C07313=1137.764,345.073,-80.303,-176.559,9.353,148.899
C07314=1137.768,344.825,-80.268,-176.562,9.349,148.898
C07315=1137.772,344.578,-80.235,-176.564,9.345,148.898
C07316=1137.777,344.331,-80.200,-176.567,9.341,148.898
C07317=1137.780,344.083,-80.166,-176.569,9.337,148.897
C07318=1137.784,343.836,-80.131,-176.572,9.333,148.897
C07319=1137.788,343.588,-80.097,-176.574,9.329,148.897
C07320=1137.792,343.340,-80.063,-176.577,9.325,148.896
C07321=1137.796,343.092,-80.029,-176.579,9.321,148.896
C07322=1137.800,342.844,-79.995,-176.582,9.318,148.896
C07323=1137.805,342.597,-79.960,-176.584,9.313,148.895
C07324=1137.808,342.349,-79.926,-176.587,9.309,148.895
C07325=1137.813,342.102,-79.891,-176.590,9.305,148.895
C07326=1137.816,341.854,-79.857,-176.592,9.301,148.894
C07327=1137.820,341.607,-79.823,-176.595,9.297,148.894
C07328=1137.825,341.359,-79.790,-176.597,9.293,148.894
C07329=1137.828,341.111,-79.755,-176.600,9.290,148.893
C07330=1137.832,340.864,-79.721,-176.602,9.285,148.893
C07331=1137.836,340.617,-79.687,-176.605,9.281,148.893
C07332=1137.840,340.368,-79.652,-176.607,9.278,148.892
C07333=1137.844,340.121,-79.619,-176.610,9.274,148.892
C07334=1137.849,339.873,-79.585,-176.613,9.270,148.892
C07335=1137.852,339.625,-79.550,-176.615,9.266,148.891
C07336=1137.857,339.345,-79.512,-176.618,9.261,148.891
C07337=1137.862,339.064,-79.473,-176.621,9.257,148.891
C07338=1137.866,338.783,-79.435,-176.624,9.253,148.891
C07339=1137.870,338.502,-79.396,-176.626,9.248,148.890
C07340=1137.875,338.255,-79.363,-176.629,9.244,148.890
C07341=1137.878,338.007,-79.329,-176.632,9.240,148.890
C07342=1137.882,337.759,-79.294,-176.634,9.237,148.889
C07343=1137.887,337.512,-79.261,-176.637,9.233,148.889
C07344=1137.890,337.265,-79.227,-176.640,9.228,148.889
C07345=1137.894,337.016,-79.194,-176.642,9.225,148.888
C07346=1137.899,336.769,-79.159,-176.645,9.221,148.888
C07347=1137.903,336.521,-79.126,-176.648,9.217,148.888
C07348=1137.906,336.274,-79.092,-176.650,9.213,148.887
C07349=1137.910,336.025,-79.059,-176.653,9.209,148.887
C07350=1137.915,335.778,-79.024,-176.655,9.206,148.887
C07351=1137.919,335.530,-78.991,-176.658,9.201,148.887
C07352=1137.923,335.283,-78.957,-176.660,9.197,148.886
C07353=1137.926,335.035,-78.924,-176.663,9.194,148.886
C07354=1137.930,334.788,-78.890,-176.665,9.190,148.886
C07355=1137.935,334.540,-78.856,-176.668,9.186,148.885
C07356=1137.939,334.292,-78.822,-176.671,9.182,148.885
C07357=1137.942,334.044,-78.789,-176.673,9.178,148.885
C07358=1137.946,333.796,-78.755,-176.676,9.174,148.885
C07359=1137.950,333.549,-78.722,-176.678,9.171,148.884
C07360=1137.954,333.301,-78.688,-176.681,9.166,148.884
C07361=1137.959,333.053,-78.655,-176.683,9.163,148.884
C07362=1137.962,332.806,-78.620,-176.686,9.159,148.884
C07363=1137.967,332.558,-78.587,-176.689,9.155,148.883
C07364=1137.971,332.310,-78.554,-176.691,9.151,148.883
C07365=1137.975,332.062,-78.521,-176.694,9.147,148.883
C07366=1137.979,331.815,-78.487,-176.696,9.144,148.882
C07367=1137.982,331.567,-78.454,-176.699,9.140,148.882
C07368=1137.986,331.319,-78.420,-176.702,9.136,148.882
C07369=1137.990,331.071,-78.387,-176.704,9.132,148.882
C07370=1137.994,330.824,-78.353,-176.707,9.128,148.881
C07371=1137.998,330.577,-78.320,-176.709,9.125,148.881
C07372=1138.003,330.329,-78.287,-176.712,9.121,148.881
C07373=1138.007,330.081,-78.254,-176.715,9.117,148.880
C07374=1138.011,329.832,-78.220,-176.717,9.113,148.880
C07375=1138.015,329.585,-78.187,-176.720,9.109,148.880
C07376=1138.019,329.337,-78.153,-176.722,9.106,148.880
C07377=1138.023,329.089,-78.120,-176.725,9.102,148.879
C07378=1138.027,328.842,-78.088,-176.728,9.098,148.879
C07379=1138.031,328.595,-78.054,-176.730,9.094,148.879
C07380=1138.035,328.347,-78.021,-176.733,9.090,148.879
C07381=1138.039,328.099,-77.988,-176.735,9.087,148.878
C07382=1138.043,327.851,-77.954,-176.738,9.083,148.878
C07383=1138.047,327.604,-77.921,-176.740,9.079,148.878
C07384=1138.051,327.356,-77.888,-176.743,9.075,148.878
C07385=1138.055,327.108,-77.855,-176.746,9.071,148.877
C07386=1138.059,326.859,-77.822,-176.749,9.068,148.877
C07387=1138.063,326.612,-77.789,-176.751,9.063,148.877
C07388=1138.068,326.364,-77.756,-176.753,9.060,148.877
C07389=1138.072,326.116,-77.723,-176.756,9.056,148.876
C07390=1138.076,325.868,-77.690,-176.759,9.053,148.876
C07391=1138.079,325.621,-77.657,-176.762,9.049,148.876
C07392=1138.083,325.373,-77.624,-176.765,9.045,148.876
C07393=1138.088,325.125,-77.591,-176.767,9.042,148.876
C07394=1138.092,324.878,-77.557,-176.769,9.037,148.875
C07395=1138.096,324.629,-77.525,-176.772,9.034,148.875
C07396=1138.100,324.382,-77.492,-176.775,9.030,148.875
C07397=1138.104,324.134,-77.459,-176.777,9.027,148.875
C07398=1138.108,323.886,-77.426,-176.780,9.022,148.874
C07399=1138.112,323.638,-77.394,-176.782,9.019,148.874
C07400=1138.116,323.390,-77.361,-176.785,9.015,148.874
C07401=1138.120,323.143,-77.328,-176.788,9.011,148.874
C07402=1138.124,322.895,-77.295,-176.790,9.008,148.873
C07403=1138.128,322.647,-77.262,-176.793,9.003,148.873
C07404=1138.132,322.399,-77.229,-176.795,9.000,148.873
C07405=1138.136,322.152,-77.197,-176.798,8.996,148.873
C07406=1138.140,321.903,-77.164,-176.801,8.993,148.872
C07407=1138.144,321.656,-77.131,-176.804,8.989,148.872
C07408=1138.148,321.408,-77.099,-176.806,8.986,148.872
C07409=1138.153,321.161,-77.066,-176.809,8.981,148.872
C07410=1138.157,320.913,-77.033,-176.811,8.978,148.872
C07411=1138.161,320.665,-77.001,-176.814,8.974,148.871
C07412=1138.165,320.417,-76.968,-176.816,8.971,148.871
C07413=1138.169,320.169,-76.935,-176.819,8.967,148.871
C07414=1138.173,319.921,-76.903,-176.822,8.964,148.871
C07415=1138.177,319.674,-76.870,-176.825,8.959,148.871
C07416=1138.181,319.425,-76.838,-176.827,8.956,148.870
C07417=1138.185,319.178,-76.805,-176.830,8.952,148.870
C07418=1138.189,318.929,-76.773,-176.832,8.949,148.870
C07419=1138.193,318.682,-76.740,-176.835,8.945,148.870
C07420=1138.198,318.434,-76.708,-176.838,8.940,148.869
C07421=1138.201,318.186,-76.676,-176.840,8.937,148.869
C07422=1138.205,317.939,-76.643,-176.843,8.933,148.869
C07423=1138.210,317.690,-76.611,-176.845,8.930,148.869
C07424=1138.213,317.443,-76.578,-176.848,8.926,148.869
C07425=1138.218,317.195,-76.546,-176.851,8.923,148.868
C07426=1138.221,316.947,-76.514,-176.854,8.918,148.868
C07427=1138.226,316.699,-76.481,-176.856,8.915,148.868
C07428=1138.230,316.451,-76.449,-176.859,8.911,148.868
C07429=1138.234,316.203,-76.417,-176.862,8.908,148.868
C07430=1138.238,315.956,-76.384,-176.864,8.904,148.867
C07431=1138.242,315.707,-76.352,-176.867,8.901,148.867
C07432=1138.246,315.460,-76.320,-176.869,8.898,148.867
C07433=1138.251,315.212,-76.287,-176.872,8.894,148.867
C07434=1138.254,314.964,-76.255,-176.874,8.890,148.867
C07435=1138.259,314.716,-76.223,-176.877,8.886,148.867
C07436=1138.262,314.468,-76.191,-176.880,8.883,148.866
C07437=1138.267,314.220,-76.159,-176.883,8.879,148.866
C07438=1138.271,313.973,-76.126,-176.885,8.876,148.866
C07439=1138.275,313.725,-76.094,-176.888,8.872,148.866
C07440=1138.280,313.447,-76.058,-176.891,8.867,148.865
C07441=1138.284,313.169,-76.023,-176.894,8.863,148.865
C07442=1138.289,312.890,-75.987,-176.897,8.859,148.865
C07443=1138.294,312.612,-75.951,-176.900,8.855,148.865
C07444=1138.298,312.364,-75.919,-176.902,8.852,148.865
C07445=1138.302,312.117,-75.887,-176.905,8.848,148.864
C07446=1138.306,311.869,-75.854,-176.908,8.845,148.864
C07447=1138.310,311.621,-75.822,-176.911,8.841,148.864
C07448=1138.313,311.373,-75.790,-176.913,8.838,148.864
C07449=1138.318,311.126,-75.758,-176.916,8.834,148.864
C07450=1138.322,310.877,-75.727,-176.918,8.830,148.864
C07451=1138.326,310.629,-75.695,-176.921,8.826,148.863
C07452=1138.331,310.382,-75.663,-176.924,8.823,148.863
C07453=1138.335,310.134,-75.631,-176.926,8.819,148.863
C07454=1138.339,309.885,-75.600,-176.929,8.816,148.863
C07455=1138.343,309.638,-75.568,-176.932,8.813,148.863
C07456=1138.347,309.389,-75.536,-176.935,8.809,148.863
C07457=1138.351,309.141,-75.504,-176.937,8.805,148.862
C07458=1138.355,308.894,-75.472,-176.940,8.801,148.862
C07459=1138.359,308.646,-75.441,-176.942,8.798,148.862
C07460=1138.364,308.398,-75.408,-176.945,8.794,148.862
C07461=1138.368,308.150,-75.377,-176.947,8.791,148.862
C07462=1138.372,307.902,-75.345,-176.950,8.788,148.862
C07463=1138.376,307.654,-75.314,-176.953,8.784,148.861
C07464=1138.380,307.406,-75.282,-176.955,8.781,148.861
C07465=1138.384,307.158,-75.250,-176.958,8.776,148.861
C07466=1138.389,306.911,-75.218,-176.961,8.773,148.861
C07467=1138.393,306.662,-75.187,-176.964,8.769,148.861
C07468=1138.397,306.415,-75.156,-176.966,8.766,148.861
C07469=1138.401,306.167,-75.124,-176.969,8.763,148.861
C07470=1138.405,305.918,-75.093,-176.972,8.759,148.860
C07471=1138.409,305.671,-75.061,-176.974,8.756,148.860
C07472=1138.413,305.422,-75.029,-176.977,8.752,148.860
C07473=1138.418,305.175,-74.997,-176.980,8.749,148.860
C07474=1138.422,304.926,-74.966,-176.983,8.745,148.860
C07475=1138.426,304.679,-74.935,-176.985,8.741,148.860
C07476=1138.430,304.430,-74.904,-176.987,8.738,148.859
C07477=1138.434,304.183,-74.872,-176.990,8.734,148.859
C07478=1138.438,303.935,-74.840,-176.993,8.731,148.859
C07479=1138.443,303.687,-74.809,-176.996,8.727,148.859
C07480=1138.446,303.439,-74.778,-176.998,8.724,148.859
C07481=1138.451,303.191,-74.747,-177.001,8.720,148.859
C07482=1138.455,302.943,-74.715,-177.004,8.717,148.859
C07483=1138.459,302.695,-74.684,-177.006,8.713,148.858
C07484=1138.463,302.447,-74.652,-177.009,8.709,148.858
C07485=1138.468,302.199,-74.622,-177.012,8.706,148.858
C07486=1138.471,301.951,-74.590,-177.014,8.703,148.858
C07487=1138.476,301.703,-74.559,-177.017,8.699,148.858
C07488=1138.480,301.455,-74.527,-177.020,8.696,148.858
C07489=1138.484,301.207,-74.496,-177.023,8.692,148.858
C07490=1138.488,300.958,-74.465,-177.025,8.689,148.858
C07491=1138.493,300.711,-74.434,-177.028,8.686,148.857
C07492=1138.497,300.462,-74.403,-177.031,8.682,148.857
C07493=1138.501,300.215,-74.371,-177.033,8.678,148.857
C07494=1138.505,299.966,-74.340,-177.036,8.675,148.857
C07495=1138.510,299.718,-74.309,-177.039,8.671,148.857
C07496=1138.513,299.470,-74.277,-177.041,8.668,148.857
C07497=1138.518,299.222,-74.247,-177.045,8.664,148.857
C07498=1138.522,298.975,-74.216,-177.047,8.661,148.856
C07499=1138.525,298.727,-74.185,-177.049,8.658,148.856
C07500=1138.530,298.479,-74.154,-177.053,8.654,148.856
C07501=1138.534,298.230,-74.123,-177.055,8.651,148.856
C07502=1138.539,297.982,-74.092,-177.057,8.648,148.856
C07503=1138.543,297.735,-74.061,-177.060,8.643,148.856
C07504=1138.546,297.486,-74.030,-177.063,8.641,148.856
C07505=1138.551,297.238,-73.999,-177.066,8.636,148.856
C07506=1138.555,296.990,-73.968,-177.068,8.633,148.855
C07507=1138.559,296.742,-73.937,-177.071,8.630,148.855
C07508=1138.564,296.494,-73.907,-177.074,8.626,148.855
C07509=1138.567,296.246,-73.875,-177.076,8.623,148.855
C07510=1138.572,295.998,-73.845,-177.079,8.620,148.855
C07511=1138.576,295.750,-73.814,-177.082,8.616,148.855
C07512=1138.580,295.501,-73.783,-177.085,8.613,148.855
C07513=1138.584,295.254,-73.752,-177.087,8.610,148.855
C07514=1138.589,295.006,-73.722,-177.090,8.606,148.855
C07515=1138.593,294.757,-73.691,-177.093,8.603,148.855
C07516=1138.597,294.510,-73.660,-177.095,8.600,148.854
C07517=1138.601,294.262,-73.630,-177.098,8.595,148.854
C07518=1138.605,294.013,-73.599,-177.101,8.593,148.854
C07519=1138.610,293.765,-73.568,-177.103,8.589,148.854
C07520=1138.614,293.517,-73.538,-177.106,8.585,148.854
C07521=1138.618,293.269,-73.506,-177.109,8.582,148.854
C07522=1138.622,293.021,-73.476,-177.111,8.579,148.854
C07523=1138.626,292.773,-73.446,-177.115,8.575,148.854
C07524=1138.630,292.524,-73.414,-177.117,8.572,148.854
C07525=1138.634,292.277,-73.384,-177.119,8.569,148.853
C07526=1138.639,292.029,-73.353,-177.123,8.565,148.853
C07527=1138.643,291.781,-73.323,-177.125,8.562,148.853
C07528=1138.647,291.533,-73.292,-177.128,8.559,148.853
C07529=1138.652,291.284,-73.262,-177.131,8.555,148.853
C07530=1138.655,291.036,-73.232,-177.134,8.552,148.853
C07531=1138.660,290.788,-73.201,-177.136,8.549,148.853
C07532=1138.663,290.540,-73.171,-177.139,8.545,148.853
C07533=1138.668,290.292,-73.140,-177.142,8.542,148.853
C07534=1138.673,290.044,-73.109,-177.144,8.538,148.853
C07535=1138.677,289.796,-73.080,-177.147,8.535,148.853
C07536=1138.681,289.547,-73.049,-177.150,8.531,148.852
C07537=1138.685,289.299,-73.018,-177.152,8.528,148.853
C07538=1138.689,289.052,-72.988,-177.155,8.525,148.852
C07539=1138.693,288.803,-72.958,-177.158,8.521,148.852
C07540=1138.698,288.555,-72.927,-177.161,8.518,148.852
C07541=1138.701,288.307,-72.897,-177.163,8.515,148.852
C07542=1138.706,288.058,-72.867,-177.166,8.511,148.852
C07543=1138.710,287.811,-72.837,-177.169,8.508,148.852
C07544=1138.714,287.535,-72.803,-177.172,8.504,148.852
C07545=1138.720,287.260,-72.770,-177.174,8.501,148.852
C07546=1138.724,286.984,-72.736,-177.178,8.497,148.852
C07547=1138.729,286.709,-72.702,-177.181,8.493,148.852
C07548=1138.733,286.460,-72.672,-177.183,8.490,148.852
C07549=1138.737,286.212,-72.642,-177.186,8.486,148.851
C07550=1138.742,285.964,-72.612,-177.189,8.483,148.851
C07551=1138.746,285.716,-72.582,-177.191,8.480,148.851
C07552=1138.750,285.468,-72.552,-177.194,8.477,148.851
C07553=1138.754,285.220,-72.522,-177.197,8.473,148.851
C07554=1138.759,284.972,-72.492,-177.200,8.470,148.851
C07555=1138.763,284.724,-72.462,-177.202,8.467,148.851
C07556=1138.767,284.475,-72.432,-177.205,8.464,148.851
C07557=1138.771,284.227,-72.402,-177.208,8.460,148.851
C07558=1138.775,283.979,-72.371,-177.211,8.457,148.851
C07559=1138.780,283.730,-72.342,-177.213,8.454,148.851
C07560=1138.784,283.483,-72.312,-177.217,8.450,148.851
C07561=1138.788,283.234,-72.282,-177.219,8.447,148.851
C07562=1138.792,282.986,-72.252,-177.222,8.444,148.851
C07563=1138.797,282.738,-72.222,-177.224,8.440,148.850
C07564=1138.801,282.490,-72.192,-177.227,8.437,148.850
C07565=1138.805,282.242,-72.162,-177.230,8.434,148.850
C07566=1138.810,281.994,-72.133,-177.233,8.430,148.850
C07567=1138.814,281.745,-72.103,-177.235,8.428,148.850
C07568=1138.818,281.497,-72.072,-177.238,8.423,148.850
C07569=1138.822,281.249,-72.043,-177.241,8.421,148.850
C07570=1138.827,281.001,-72.013,-177.243,8.417,148.850
C07571=1138.831,280.753,-71.984,-177.246,8.414,148.850
C07572=1138.835,280.505,-71.954,-177.249,8.410,148.850
C07573=1138.840,280.256,-71.924,-177.252,8.407,148.850
C07574=1138.844,280.008,-71.894,-177.255,8.404,148.850
C07575=1138.848,279.760,-71.865,-177.257,8.401,148.850
C07576=1138.852,279.512,-71.835,-177.260,8.397,148.850
C07577=1138.856,279.264,-71.805,-177.263,8.394,148.850
C07578=1138.860,279.016,-71.776,-177.265,8.391,148.850
C07579=1138.864,278.767,-71.746,-177.268,8.388,148.850
C07580=1138.869,278.519,-71.716,-177.271,8.384,148.850
C07581=1138.874,278.271,-71.687,-177.274,8.381,148.850
C07582=1138.878,278.022,-71.657,-177.276,8.378,148.850
C07583=1138.882,277.774,-71.628,-177.279,8.375,148.850
C07584=1138.886,277.526,-71.598,-177.281,8.372,148.849
C07585=1138.890,277.277,-71.569,-177.285,8.368,148.849
C07586=1138.894,277.029,-71.540,-177.288,8.365,148.849
C07587=1138.899,276.781,-71.510,-177.290,8.362,148.849
C07588=1138.903,276.533,-71.481,-177.293,8.359,148.849
C07589=1138.907,276.284,-71.451,-177.296,8.355,148.849
C07590=1138.911,276.036,-71.422,-177.298,8.352,148.849
C07591=1138.915,275.788,-71.392,-177.301,8.349,148.849
C07592=1138.920,275.540,-71.363,-177.304,8.346,148.849
C07593=1138.924,275.292,-71.334,-177.306,8.343,148.849
C07594=1138.928,275.044,-71.304,-177.310,8.339,148.849
C07595=1138.933,274.795,-71.275,-177.312,8.336,148.849
C07596=1138.937,274.547,-71.245,-177.315,8.333,148.849
C07597=1138.941,274.299,-71.216,-177.318,8.330,148.849
C07598=1138.945,274.051,-71.186,-177.320,8.327,148.849
C07599=1138.949,273.802,-71.157,-177.323,8.323,148.849
C07600=1138.954,273.554,-71.129,-177.326,8.320,148.849
C07601=1138.959,273.306,-71.099,-177.329,8.317,148.849
C07602=1138.963,273.058,-71.070,-177.331,8.314,148.849
C07603=1138.967,272.809,-71.040,-177.334,8.311,148.849
C07604=1138.971,272.561,-71.011,-177.337,8.307,148.849
C07605=1138.976,272.312,-70.982,-177.340,8.304,148.849
C07606=1138.979,272.064,-70.953,-177.342,8.301,148.849
C07607=1138.984,271.817,-70.924,-177.345,8.298,148.849
C07608=1138.988,271.568,-70.895,-177.348,8.295,148.849
C07609=1138.993,271.320,-70.866,-177.351,8.291,148.849
C07610=1138.997,271.071,-70.836,-177.354,8.288,148.849
C07611=1139.001,270.823,-70.807,-177.356,8.285,148.849
C07612=1139.006,270.575,-70.779,-177.359,8.282,148.849
C07613=1139.009,270.327,-70.750,-177.361,8.279,148.849
C07614=1139.014,270.079,-70.720,-177.364,8.276,148.849
C07615=1139.018,269.830,-70.692,-177.368,8.272,148.849
C07616=1139.023,269.582,-70.663,-177.370,8.269,148.849
C07617=1139.027,269.333,-70.634,-177.373,8.266,148.849
C07618=1139.031,269.085,-70.605,-177.376,8.263,148.849
C07619=1139.035,268.837,-70.575,-177.378,8.260,148.849
C07620=1139.040,268.589,-70.547,-177.381,8.257,148.849
C07621=1139.044,268.341,-70.518,-177.384,8.253,148.849
C07622=1139.048,268.092,-70.489,-177.386,8.250,148.848
C07623=1139.052,267.844,-70.460,-177.389,8.247,148.849
C07624=1139.057,267.596,-70.432,-177.392,8.244,148.849
C07625=1139.062,267.347,-70.402,-177.395,8.241,148.849
C07626=1139.065,267.099,-70.374,-177.397,8.238,148.849
C07627=1139.070,266.851,-70.345,-177.400,8.234,148.849
C07628=1139.075,266.602,-70.316,-177.403,8.231,148.849
C07629=1139.078,266.354,-70.287,-177.406,8.228,148.849
C07630=1139.082,266.105,-70.259,-177.408,8.225,148.849
C07631=1139.088,265.857,-70.230,-177.411,8.222,148.849
C07632=1139.091,265.609,-70.201,-177.414,8.219,148.849
C07633=1139.095,265.360,-70.173,-177.417,8.216,148.849
C07634=1139.101,265.112,-70.144,-177.420,8.212,148.848
C07635=1139.104,264.864,-70.115,-177.422,8.209,148.849
C07636=1139.109,264.615,-70.087,-177.425,8.206,148.849
C07637=1139.113,264.368,-70.059,-177.428,8.204,148.849
C07638=1139.117,264.119,-70.029,-177.430,8.200,148.849
C07639=1139.122,263.871,-70.001,-177.433,8.197,148.849
C07640=1139.126,263.622,-69.973,-177.436,8.194,148.849
C07641=1139.130,263.374,-69.944,-177.439,8.191,148.849
C07642=1139.134,263.126,-69.916,-177.442,8.187,148.849
C07643=1139.139,262.877,-69.887,-177.445,8.185,148.849
C07644=1139.143,262.629,-69.858,-177.447,8.182,148.849
C07645=1139.147,262.381,-69.830,-177.450,8.179,148.849
C07646=1139.152,262.132,-69.801,-177.452,8.175,148.849
C07647=1139.156,261.885,-69.773,-177.455,8.173,148.849
C07648=1139.161,261.610,-69.742,-177.459,8.169,148.849
C07649=1139.166,261.337,-69.711,-177.461,8.166,148.849
C07650=1139.171,261.064,-69.679,-177.465,8.162,148.849
C07651=1139.175,260.790,-69.648,-177.468,8.159,148.849
C07652=1139.180,260.542,-69.620,-177.471,8.155,148.849
C07653=1139.184,260.293,-69.591,-177.473,8.152,148.849
C07654=1139.188,260.045,-69.564,-177.476,8.149,148.849
C07655=1139.193,259.796,-69.535,-177.479,8.146,148.849
C07656=1139.197,259.548,-69.507,-177.482,8.143,148.849
C07657=1139.201,259.300,-69.478,-177.484,8.141,148.849
C07658=1139.206,259.052,-69.451,-177.487,8.137,148.849
C07659=1139.210,258.803,-69.422,-177.490,8.134,148.849
C07660=1139.214,258.554,-69.394,-177.492,8.131,148.849
C07661=1139.218,258.306,-69.366,-177.496,8.128,148.849
C07662=1139.223,258.057,-69.337,-177.499,8.125,148.849
C07663=1139.227,257.810,-69.309,-177.501,8.122,148.849
C07664=1139.231,257.561,-69.281,-177.504,8.119,148.849
C07665=1139.236,257.313,-69.253,-177.507,8.116,148.849
C07666=1139.240,257.064,-69.225,-177.509,8.113,148.849
C07667=1139.244,256.816,-69.197,-177.512,8.110,148.849
C07668=1139.249,256.568,-69.169,-177.515,8.107,148.849
C07669=1139.253,256.320,-69.140,-177.517,8.104,148.849
C07670=1139.258,256.071,-69.113,-177.520,8.101,148.849
C07671=1139.262,255.822,-69.085,-177.523,8.098,148.849
C07672=1139.266,255.574,-69.057,-177.526,8.095,148.849
C07673=1139.270,255.326,-69.029,-177.529,8.091,148.849
C07674=1139.275,255.078,-69.000,-177.532,8.088,148.849
C07675=1139.279,254.829,-68.972,-177.535,8.085,148.849
C07676=1139.284,254.580,-68.945,-177.537,8.082,148.849
C07677=1139.288,254.333,-68.917,-177.540,8.079,148.849
C07678=1139.293,254.084,-68.889,-177.543,8.076,148.849
C07679=1139.297,253.836,-68.861,-177.545,8.073,148.850
C07680=1139.301,253.587,-68.833,-177.548,8.070,148.850
C07681=1139.305,253.339,-68.806,-177.551,8.068,148.850
C07682=1139.309,253.090,-68.778,-177.554,8.065,148.850
C07683=1139.314,252.841,-68.750,-177.557,8.062,148.850
C07684=1139.319,252.594,-68.722,-177.559,8.058,148.850
C07685=1139.323,252.345,-68.694,-177.562,8.056,148.850
C07686=1139.327,252.096,-68.667,-177.564,8.053,148.850
C07687=1139.332,251.849,-68.639,-177.567,8.050,148.850
C07688=1139.336,251.599,-68.612,-177.571,8.046,148.850
C07689=1139.341,251.351,-68.583,-177.573,8.043,148.850
C07690=1139.344,251.103,-68.555,-177.576,8.040,148.850
C07691=1139.349,250.854,-68.528,-177.579,8.037,148.850
C07692=1139.353,250.606,-68.500,-177.582,8.034,148.850
C07693=1139.358,250.357,-68.473,-177.584,8.031,148.850
C07694=1139.362,250.109,-68.445,-177.587,8.028,148.850
C07695=1139.367,249.861,-68.418,-177.590,8.025,148.850
C07696=1139.370,249.612,-68.390,-177.593,8.022,148.850
C07697=1139.375,249.364,-68.363,-177.595,8.019,148.850
C07698=1139.379,249.116,-68.335,-177.598,8.016,148.850
C07699=1139.383,248.867,-68.308,-177.601,8.014,148.851
C07700=1139.388,248.619,-68.280,-177.604,8.011,148.851
C07701=1139.392,248.370,-68.253,-177.607,8.008,148.851
C07702=1139.397,248.122,-68.224,-177.609,8.005,148.851
C07703=1139.401,247.873,-68.197,-177.612,8.002,148.851
C07704=1139.406,247.624,-68.170,-177.615,7.999,148.851
C07705=1139.410,247.376,-68.142,-177.617,7.996,148.851
C07706=1139.415,247.128,-68.115,-177.620,7.993,148.851
C07707=1139.419,246.879,-68.088,-177.623,7.990,148.851
C07708=1139.423,246.631,-68.061,-177.626,7.987,148.851
C07709=1139.427,246.383,-68.033,-177.628,7.984,148.851
C07710=1139.432,246.133,-68.006,-177.631,7.981,148.851
C07711=1139.436,245.886,-67.978,-177.634,7.978,148.851
C07712=1139.441,245.637,-67.951,-177.637,7.975,148.851
C07713=1139.445,245.389,-67.924,-177.640,7.972,148.851
C07714=1139.450,245.140,-67.897,-177.642,7.969,148.851
C07715=1139.454,244.891,-67.869,-177.645,7.967,148.851
C07716=1139.458,244.643,-67.842,-177.648,7.964,148.852
C07717=1139.463,244.395,-67.815,-177.651,7.961,148.852
C07718=1139.468,244.146,-67.788,-177.654,7.958,148.852
C07719=1139.472,243.898,-67.761,-177.656,7.955,148.852
C07720=1139.475,243.649,-67.733,-177.659,7.952,148.852
C07721=1139.480,243.401,-67.706,-177.662,7.949,148.852
C07722=1139.485,243.152,-67.679,-177.665,7.946,148.852
C07723=1139.489,242.904,-67.652,-177.668,7.943,148.852
C07724=1139.494,242.655,-67.625,-177.670,7.940,148.852
C07725=1139.498,242.406,-67.597,-177.673,7.937,148.852
C07726=1139.502,242.158,-67.571,-177.676,7.934,148.852
C07727=1139.506,241.909,-67.544,-177.679,7.932,148.852
C07728=1139.511,241.662,-67.516,-177.682,7.929,148.853
C07729=1139.516,241.413,-67.489,-177.684,7.926,148.853
C07730=1139.520,241.165,-67.462,-177.687,7.923,148.853
C07731=1139.524,240.916,-67.436,-177.690,7.920,148.853
C07732=1139.528,240.667,-67.408,-177.693,7.917,148.853
C07733=1139.533,240.419,-67.381,-177.696,7.914,148.853
C07734=1139.537,240.170,-67.354,-177.698,7.911,148.853
C07735=1139.541,239.922,-67.328,-177.701,7.908,148.853
C07736=1139.546,239.673,-67.301,-177.704,7.905,148.853
C07737=1139.551,239.424,-67.274,-177.707,7.902,148.853
C07738=1139.555,239.176,-67.248,-177.710,7.900,148.853
C07739=1139.560,238.928,-67.221,-177.712,7.897,148.853
C07740=1139.564,238.679,-67.194,-177.715,7.894,148.853
C07741=1139.568,238.431,-67.167,-177.718,7.891,148.854
C07742=1139.573,238.183,-67.140,-177.721,7.888,148.854
C07743=1139.577,237.933,-67.113,-177.724,7.885,148.854
C07744=1139.581,237.685,-67.086,-177.726,7.882,148.854
C07745=1139.586,237.436,-67.060,-177.729,7.879,148.854
C07746=1139.590,237.187,-67.033,-177.732,7.876,148.854
C07747=1139.594,236.939,-67.006,-177.735,7.873,148.854
C07748=1139.599,236.691,-66.979,-177.738,7.870,148.854
C07749=1139.604,236.442,-66.952,-177.740,7.867,148.854
C07750=1139.608,236.194,-66.926,-177.743,7.865,148.854
C07751=1139.613,235.945,-66.899,-177.746,7.862,148.854
C07752=1139.618,235.673,-66.870,-177.749,7.859,148.854
C07753=1139.622,235.402,-66.841,-177.752,7.856,148.855
C07754=1139.627,235.129,-66.812,-177.754,7.853,148.855
C07755=1139.632,234.858,-66.783,-177.758,7.850,148.855
C07756=1139.636,234.609,-66.756,-177.761,7.847,148.855
C07757=1139.641,234.360,-66.730,-177.764,7.844,148.855
C07758=1139.645,234.112,-66.704,-177.767,7.841,148.855
C07759=1139.649,233.864,-66.677,-177.769,7.838,148.855
C07760=1139.654,233.615,-66.651,-177.772,7.836,148.855
C07761=1139.658,233.366,-66.624,-177.774,7.833,148.855
C07762=1139.663,233.118,-66.598,-177.777,7.830,148.856
C07763=1139.667,232.869,-66.571,-177.780,7.827,148.856
C07764=1139.671,232.621,-66.544,-177.783,7.824,148.856
C07765=1139.676,232.372,-66.518,-177.786,7.821,148.856
C07766=1139.680,232.124,-66.492,-177.788,7.818,148.856
C07767=1139.685,231.874,-66.465,-177.791,7.815,148.856
C07768=1139.689,231.626,-66.439,-177.794,7.812,148.856
C07769=1139.694,231.378,-66.413,-177.797,7.810,148.856
C07770=1139.698,231.130,-66.386,-177.800,7.807,148.856
C07771=1139.703,230.881,-66.361,-177.803,7.804,148.856
C07772=1139.707,230.632,-66.334,-177.805,7.802,148.857
C07773=1139.711,230.384,-66.308,-177.808,7.799,148.857
C07774=1139.716,230.135,-66.282,-177.811,7.796,148.857
C07775=1139.720,229.886,-66.255,-177.814,7.793,148.857
C07776=1139.725,229.637,-66.229,-177.816,7.790,148.857
C07777=1139.729,229.389,-66.202,-177.819,7.787,148.857
C07778=1139.734,229.141,-66.177,-177.822,7.785,148.857
C07779=1139.738,228.892,-66.151,-177.825,7.782,148.857
C07780=1139.743,228.644,-66.124,-177.828,7.779,148.858
C07781=1139.747,228.395,-66.098,-177.831,7.776,148.858
C07782=1139.751,228.146,-66.072,-177.833,7.774,148.858
C07783=1139.756,227.897,-66.045,-177.836,7.771,148.858
C07784=1139.760,227.649,-66.020,-177.839,7.768,148.858
C07785=1139.765,227.401,-65.994,-177.841,7.765,148.858
C07786=1139.769,227.152,-65.968,-177.844,7.762,148.858
C07787=1139.774,226.903,-65.941,-177.847,7.760,148.858
C07788=1139.778,226.654,-65.916,-177.850,7.757,148.858
C07789=1139.782,226.406,-65.890,-177.853,7.754,148.859
C07790=1139.786,226.157,-65.863,-177.856,7.751,148.859
C07791=1139.792,225.909,-65.838,-177.858,7.749,148.859
C07792=1139.796,225.660,-65.812,-177.861,7.746,148.859
C07793=1139.800,225.411,-65.786,-177.864,7.743,148.859
C07794=1139.805,225.163,-65.760,-177.867,7.740,148.859
C07795=1139.810,224.915,-65.734,-177.870,7.738,148.859
C07796=1139.814,224.666,-65.708,-177.873,7.735,148.859
C07797=1139.818,224.417,-65.682,-177.875,7.732,148.860
C07798=1139.823,224.168,-65.656,-177.878,7.729,148.860
C07799=1139.827,223.920,-65.631,-177.880,7.727,148.860
C07800=1139.832,223.671,-65.605,-177.883,7.724,148.860
C07801=1139.837,223.422,-65.579,-177.887,7.721,148.860
C07802=1139.841,223.174,-65.553,-177.889,7.719,148.860
C07803=1139.845,222.925,-65.527,-177.892,7.716,148.860
C07804=1139.850,222.677,-65.502,-177.895,7.713,148.860
C07805=1139.854,222.428,-65.476,-177.898,7.710,148.861
C07806=1139.858,222.179,-65.450,-177.900,7.708,148.861
C07807=1139.863,221.931,-65.425,-177.903,7.705,148.861
C07808=1139.867,221.682,-65.399,-177.906,7.702,148.861
C07809=1139.872,221.433,-65.374,-177.909,7.699,148.861
C07810=1139.876,221.185,-65.348,-177.912,7.696,148.861
C07811=1139.881,220.936,-65.322,-177.914,7.694,148.861
C07812=1139.886,220.687,-65.296,-177.917,7.692,148.862
C07813=1139.890,220.439,-65.270,-177.920,7.689,148.862
C07814=1139.895,220.190,-65.245,-177.923,7.686,148.862
C07815=1139.899,219.942,-65.219,-177.926,7.683,148.862
C07816=1139.903,219.693,-65.193,-177.928,7.680,148.862
C07817=1139.908,219.445,-65.168,-177.932,7.678,148.862
C07818=1139.912,219.195,-65.143,-177.934,7.675,148.862
C07819=1139.917,218.946,-65.117,-177.937,7.673,148.863
C07820=1139.921,218.698,-65.092,-177.939,7.670,148.863
C07821=1139.926,218.450,-65.066,-177.942,7.667,148.863
C07822=1139.930,218.201,-65.041,-177.945,7.664,148.863
C07823=1139.935,217.952,-65.016,-177.948,7.662,148.863
C07824=1139.939,217.704,-64.991,-177.951,7.659,148.863
C07825=1139.943,217.455,-64.965,-177.953,7.656,148.863
C07826=1139.948,217.207,-64.939,-177.956,7.653,148.864
C07827=1139.952,216.957,-64.914,-177.959,7.651,148.864
C07828=1139.957,216.709,-64.889,-177.962,7.648,148.864
C07829=1139.961,216.460,-64.863,-177.964,7.646,148.864
C07830=1139.966,216.212,-64.838,-177.967,7.643,148.864
C07831=1139.970,215.963,-64.813,-177.970,7.640,148.864
C07832=1139.975,215.714,-64.787,-177.973,7.637,148.865
C07833=1139.980,215.466,-64.762,-177.976,7.635,148.865
C07834=1139.983,215.217,-64.737,-177.978,7.632,148.865
C07835=1139.988,214.969,-64.712,-177.982,7.630,148.865
C07836=1139.993,214.719,-64.687,-177.984,7.627,148.865
C07837=1139.998,214.471,-64.661,-177.987,7.624,148.865
C07838=1140.002,214.222,-64.636,-177.989,7.622,148.865
C07839=1140.007,213.974,-64.611,-177.993,7.619,148.866
C07840=1140.010,213.725,-64.586,-177.996,7.617,148.866
C07841=1140.015,213.476,-64.561,-177.998,7.614,148.866
C07842=1140.020,213.228,-64.535,-178.001,7.611,148.866
C07843=1140.024,212.978,-64.510,-178.004,7.609,148.866
C07844=1140.029,212.730,-64.485,-178.007,7.606,148.866
C07845=1140.033,212.481,-64.461,-178.009,7.603,148.867
C07846=1140.038,212.233,-64.435,-178.013,7.601,148.867
C07847=1140.042,211.983,-64.410,-178.015,7.599,148.867
C07848=1140.047,211.735,-64.385,-178.018,7.596,148.867
C07849=1140.051,211.486,-64.360,-178.021,7.593,148.867
C07850=1140.056,211.238,-64.335,-178.024,7.590,148.868
C07851=1140.060,210.989,-64.310,-178.027,7.587,148.868
C07852=1140.065,210.740,-64.286,-178.029,7.585,148.868
C07853=1140.069,210.492,-64.260,-178.032,7.583,148.868
C07854=1140.074,210.243,-64.235,-178.035,7.580,148.868
C07855=1140.079,209.995,-64.210,-178.038,7.577,148.868
C07856=1140.083,209.724,-64.183,-178.041,7.574,148.869
C07857=1140.088,209.453,-64.156,-178.044,7.571,148.869
C07858=1140.093,209.183,-64.129,-178.047,7.568,148.869
C07859=1140.098,208.912,-64.102,-178.050,7.566,148.869
C07860=1140.103,208.663,-64.077,-178.053,7.563,148.869
C07861=1140.107,208.414,-64.053,-178.055,7.561,148.869
C07862=1140.111,208.166,-64.028,-178.058,7.558,148.870
C07863=1140.116,207.917,-64.003,-178.061,7.555,148.870
C07864=1140.120,207.668,-63.978,-178.064,7.553,148.870
C07865=1140.125,207.419,-63.954,-178.066,7.551,148.870
C07866=1140.129,207.170,-63.929,-178.069,7.548,148.870
C07867=1140.134,206.922,-63.904,-178.072,7.545,148.870
C07868=1140.139,206.673,-63.879,-178.075,7.543,148.871
C07869=1140.143,206.424,-63.855,-178.078,7.540,148.871
C07870=1140.148,206.176,-63.830,-178.080,7.537,148.871
C07871=1140.152,205.927,-63.806,-178.084,7.535,148.871
C07872=1140.157,205.678,-63.781,-178.086,7.533,148.871
C07873=1140.161,205.430,-63.756,-178.089,7.530,148.872
C07874=1140.166,205.181,-63.732,-178.092,7.527,148.872
C07875=1140.170,204.932,-63.707,-178.095,7.524,148.872
C07876=1140.175,204.683,-63.683,-178.097,7.523,148.872
C07877=1140.180,204.435,-63.658,-178.100,7.520,148.872
C07878=1140.184,204.186,-63.633,-178.103,7.517,148.873
C07879=1140.188,203.937,-63.609,-178.106,7.515,148.873
C07880=1140.194,203.688,-63.585,-178.109,7.512,148.873
C07881=1140.197,203.439,-63.560,-178.111,7.509,148.873
C07882=1140.203,203.191,-63.536,-178.114,7.508,148.873
C07883=1140.207,202.942,-63.511,-178.117,7.505,148.874
C07884=1140.211,202.693,-63.486,-178.120,7.502,148.874
C07885=1140.216,202.444,-63.462,-178.123,7.499,148.874
C07886=1140.220,202.196,-63.438,-178.125,7.497,148.874
C07887=1140.225,201.947,-63.414,-178.128,7.495,148.874
C07888=1140.229,201.698,-63.389,-178.131,7.492,148.875
C07889=1140.234,201.449,-63.365,-178.134,7.490,148.875
C07890=1140.239,201.201,-63.340,-178.137,7.487,148.875
C07891=1140.242,200.952,-63.316,-178.140,7.484,148.875
C07892=1140.248,200.703,-63.291,-178.142,7.482,148.875
C07893=1140.252,200.454,-63.268,-178.145,7.480,148.876
C07894=1140.257,200.206,-63.244,-178.148,7.477,148.876
C07895=1140.261,199.956,-63.219,-178.151,7.475,148.876
C07896=1140.266,199.708,-63.195,-178.153,7.472,148.876
C07897=1140.270,199.459,-63.171,-178.157,7.469,148.877
C07898=1140.275,199.211,-63.146,-178.159,7.467,148.877
C07899=1140.280,198.962,-63.123,-178.162,7.465,148.877
C07900=1140.284,198.712,-63.098,-178.165,7.462,148.877
C07901=1140.289,198.464,-63.074,-178.167,7.460,148.877
C07902=1140.293,198.215,-63.050,-178.170,7.457,148.878
C07903=1140.298,197.966,-63.026,-178.173,7.454,148.878
C07904=1140.302,197.717,-63.002,-178.176,7.453,148.878
C07905=1140.307,197.468,-62.977,-178.179,7.450,148.878
C07906=1140.311,197.220,-62.953,-178.182,7.447,148.878
C07907=1140.316,196.971,-62.930,-178.184,7.445,148.879
C07908=1140.320,196.723,-62.906,-178.187,7.442,148.879
C07909=1140.325,196.474,-62.881,-178.190,7.440,148.879
C07910=1140.330,196.224,-62.857,-178.193,7.438,148.879
C07911=1140.334,195.976,-62.833,-178.196,7.435,148.879
C07912=1140.338,195.727,-62.809,-178.198,7.433,148.880
C07913=1140.343,195.478,-62.786,-178.201,7.430,148.880
C07914=1140.347,195.230,-62.762,-178.204,7.427,148.880
C07915=1140.353,194.981,-62.738,-178.207,7.426,148.880
C07916=1140.357,194.732,-62.714,-178.210,7.423,148.881
C07917=1140.362,194.483,-62.690,-178.213,7.420,148.881
C07918=1140.366,194.234,-62.666,-178.215,7.418,148.881
C07919=1140.370,193.986,-62.642,-178.218,7.415,148.881
C07920=1140.375,193.737,-62.618,-178.221,7.414,148.881
C07921=1140.379,193.488,-62.594,-178.224,7.411,148.882
C07922=1140.385,193.239,-62.570,-178.227,7.408,148.882
C07923=1140.389,192.990,-62.546,-178.229,7.406,148.882
C07924=1140.394,192.741,-62.523,-178.232,7.403,148.882
C07925=1140.398,192.492,-62.499,-178.235,7.401,148.883
C07926=1140.403,192.244,-62.475,-178.238,7.399,148.883
C07927=1140.408,191.995,-62.452,-178.241,7.396,148.883
C07928=1140.412,191.746,-62.428,-178.243,7.394,148.883
C07929=1140.417,191.497,-62.405,-178.246,7.391,148.883
C07930=1140.420,191.248,-62.380,-178.249,7.389,148.884
C07931=1140.425,190.999,-62.357,-178.252,7.387,148.884
C07932=1140.430,190.750,-62.333,-178.255,7.384,148.884
C07933=1140.434,190.502,-62.309,-178.257,7.382,148.884
C07934=1140.439,190.253,-62.286,-178.260,7.380,148.885
C07935=1140.444,190.004,-62.263,-178.263,7.377,148.885
C07936=1140.448,189.755,-62.239,-178.266,7.375,148.885
C07937=1140.453,189.506,-62.215,-178.269,7.372,148.885
C07938=1140.457,189.257,-62.192,-178.271,7.370,148.886
C07939=1140.462,189.009,-62.168,-178.274,7.367,148.886
C07940=1140.466,188.760,-62.144,-178.278,7.365,148.886
C07941=1140.471,188.511,-62.121,-178.280,7.363,148.886
C07942=1140.476,188.262,-62.098,-178.283,7.360,148.887
C07943=1140.480,188.013,-62.074,-178.285,7.358,148.887
C07944=1140.485,187.764,-62.050,-178.289,7.356,148.887
C07945=1140.490,187.515,-62.027,-178.291,7.353,148.887
C07946=1140.494,187.266,-62.004,-178.294,7.351,148.888
C07947=1140.500,187.018,-61.981,-178.297,7.348,148.888
C07948=1140.504,186.770,-61.957,-178.300,7.346,148.888
C07949=1140.508,186.521,-61.934,-178.302,7.343,148.888
C07950=1140.513,186.272,-61.910,-178.305,7.342,148.889
C07951=1140.517,186.023,-61.887,-178.308,7.339,148.889
C07952=1140.522,185.774,-61.864,-178.311,7.337,148.889
C07953=1140.527,185.525,-61.840,-178.314,7.335,148.889
C07954=1140.532,185.276,-61.817,-178.316,7.332,148.890
C07955=1140.536,185.027,-61.794,-178.319,7.330,148.890
C07956=1140.540,184.778,-61.771,-178.322,7.327,148.890
C07957=1140.545,184.529,-61.747,-178.325,7.325,148.890
C07958=1140.549,184.280,-61.723,-178.328,7.322,148.890
C07959=1140.554,184.031,-61.700,-178.330,7.321,148.891
C07960=1140.559,183.762,-61.675,-178.334,7.318,148.891
C07961=1140.564,183.492,-61.651,-178.337,7.315,148.891
C07962=1140.569,183.222,-61.626,-178.340,7.313,148.892
C07963=1140.574,182.953,-61.600,-178.343,7.310,148.892
C07964=1140.579,182.704,-61.576,-178.345,7.308,148.892
C07965=1140.583,182.455,-61.554,-178.349,7.305,148.892
C07966=1140.588,182.206,-61.531,-178.351,7.303,148.893
C07967=1140.593,181.957,-61.508,-178.354,7.301,148.893
C07968=1140.598,181.709,-61.485,-178.357,7.299,148.893
C07969=1140.602,181.460,-61.462,-178.360,7.296,148.893
C07970=1140.607,181.211,-61.439,-178.362,7.295,148.894
C07971=1140.611,180.962,-61.415,-178.365,7.292,148.894
C07972=1140.615,180.713,-61.392,-178.368,7.290,148.894
C07973=1140.620,180.464,-61.369,-178.371,7.287,148.895
C07974=1140.625,180.215,-61.346,-178.373,7.285,148.895
C07975=1140.629,179.966,-61.324,-178.377,7.283,148.895
C07976=1140.634,179.717,-61.301,-178.379,7.281,148.895
C07977=1140.639,179.468,-61.277,-178.382,7.278,148.896
C07978=1140.643,179.220,-61.255,-178.385,7.276,148.896
C07979=1140.648,178.970,-61.231,-178.388,7.274,148.896
C07980=1140.652,178.722,-61.209,-178.390,7.272,148.896
C07981=1140.657,178.473,-61.186,-178.393,7.269,148.897
C07982=1140.662,178.224,-61.163,-178.396,7.267,148.897
C07983=1140.666,177.975,-61.140,-178.399,7.265,148.897
C07984=1140.671,177.726,-61.118,-178.401,7.263,148.897
C07985=1140.675,177.477,-61.095,-178.405,7.260,148.898
C07986=1140.680,177.228,-61.072,-178.407,7.258,148.898
C07987=1140.685,176.979,-61.049,-178.410,7.255,148.898
C07988=1140.690,176.731,-61.027,-178.413,7.254,148.899
C07989=1140.694,176.482,-61.003,-178.416,7.251,148.899
C07990=1140.699,176.232,-60.981,-178.418,7.249,148.899
C07991=1140.703,175.983,-60.958,-178.422,7.247,148.899
C07992=1140.708,175.735,-60.935,-178.424,7.244,148.900
C07993=1140.713,175.486,-60.913,-178.427,7.242,148.900
C07994=1140.717,175.237,-60.890,-178.430,7.240,148.900
C07995=1140.722,174.988,-60.868,-178.433,7.237,148.900
C07996=1140.726,174.739,-60.845,-178.435,7.236,148.901
C07997=1140.731,174.490,-60.822,-178.438,7.233,148.901
C07998=1140.735,174.241,-60.800,-178.441,7.231,148.901
C07999=1140.741,173.993,-60.777,-178.444,7.228,148.902
C08000=1140.745,173.743,-60.754,-178.447,7.226,148.902
C08001=1140.750,173.494,-60.731,-178.449,7.225,148.902
C08002=1140.755,173.246,-60.709,-178.453,7.222,148.903
C08003=1140.758,172.997,-60.687,-178.455,7.220,148.903
C08004=1140.763,172.747,-60.664,-178.458,7.217,148.903
C08005=1140.768,172.499,-60.642,-178.461,7.216,148.903
C08006=1140.773,172.249,-60.619,-178.464,7.213,148.904
C08007=1140.777,172.000,-60.597,-178.466,7.211,148.904
C08008=1140.783,171.752,-60.574,-178.470,7.209,148.904
C08009=1140.787,171.502,-60.552,-178.472,7.206,148.904
C08010=1140.791,171.254,-60.530,-178.474,7.205,148.905
C08011=1140.796,171.005,-60.507,-178.478,7.202,148.905
C08012=1140.801,170.755,-60.485,-178.480,7.200,148.905
C08013=1140.805,170.507,-60.462,-178.483,7.198,148.906
C08014=1140.810,170.258,-60.440,-178.486,7.196,148.906
C08015=1140.815,170.009,-60.418,-178.489,7.193,148.906
C08016=1140.819,169.760,-60.395,-178.492,7.191,148.907
C08017=1140.824,169.511,-60.373,-178.495,7.189,148.907
C08018=1140.829,169.262,-60.351,-178.498,7.187,148.907
C08019=1140.833,169.013,-60.328,-178.500,7.185,148.907
C08020=1140.839,168.764,-60.306,-178.503,7.182,148.908
C08021=1140.843,168.515,-60.284,-178.506,7.181,148.908
C08022=1140.847,168.266,-60.262,-178.509,7.178,148.908
C08023=1140.852,168.018,-60.239,-178.511,7.176,148.909
C08024=1140.857,167.768,-60.217,-178.514,7.174,148.909
C08025=1140.862,167.519,-60.195,-178.517,7.171,148.909
C08026=1140.866,167.270,-60.173,-178.520,7.170,148.910
C08027=1140.871,167.021,-60.151,-178.523,7.167,148.910
C08028=1140.875,166.772,-60.128,-178.526,7.166,148.910
C08029=1140.880,166.524,-60.106,-178.528,7.163,148.910
C08030=1140.885,166.274,-60.084,-178.531,7.161,148.911
C08031=1140.889,166.026,-60.063,-178.534,7.159,148.911
C08032=1140.894,165.776,-60.040,-178.537,7.156,148.911
C08033=1140.899,165.528,-60.018,-178.539,7.155,148.912
C08034=1140.904,165.278,-59.996,-178.542,7.153,148.912
C08035=1140.908,165.030,-59.974,-178.545,7.150,148.912
C08036=1140.912,164.781,-59.952,-178.548,7.148,148.913
C08037=1140.917,164.532,-59.930,-178.551,7.146,148.913
C08038=1140.922,164.283,-59.908,-178.554,7.144,148.913
C08039=1140.927,164.034,-59.886,-178.556,7.142,148.914
C08040=1140.931,163.785,-59.864,-178.559,7.139,148.914
C08041=1140.936,163.536,-59.842,-178.562,7.138,148.914
C08042=1140.940,163.287,-59.820,-178.565,7.135,148.914
C08043=1140.945,163.038,-59.798,-178.567,7.133,148.915
C08044=1140.950,162.789,-59.776,-178.570,7.131,148.915
C08045=1140.954,162.540,-59.755,-178.573,7.129,148.915
C08046=1140.959,162.291,-59.733,-178.576,7.127,148.916
C08047=1140.964,162.042,-59.711,-178.578,7.125,148.916
C08048=1140.969,161.793,-59.689,-178.582,7.123,148.916
C08049=1140.974,161.544,-59.667,-178.584,7.121,148.917
C08050=1140.978,161.295,-59.645,-178.588,7.118,148.917
C08051=1140.983,161.045,-59.624,-178.590,7.116,148.917
C08052=1140.988,160.796,-59.602,-178.592,7.114,148.918
C08053=1140.992,160.547,-59.580,-178.596,7.112,148.918
C08054=1140.997,160.298,-59.558,-178.598,7.110,148.918
C08055=1141.002,160.050,-59.536,-178.601,7.109,148.919
C08056=1141.006,159.800,-59.514,-178.604,7.106,148.919
C08057=1141.011,159.552,-59.493,-178.607,7.104,148.919
C08058=1141.016,159.303,-59.472,-178.609,7.102,148.920
C08059=1141.020,159.053,-59.450,-178.613,7.100,148.920
C08060=1141.025,158.805,-59.428,-178.615,7.098,148.920
C08061=1141.030,158.555,-59.406,-178.618,7.096,148.920
C08062=1141.034,158.307,-59.384,-178.621,7.093,148.921
C08063=1141.039,158.058,-59.364,-178.624,7.092,148.921
C08064=1141.044,157.789,-59.340,-178.627,7.089,148.922
C08065=1141.050,157.520,-59.317,-178.630,7.087,148.922
C08066=1141.054,157.250,-59.294,-178.633,7.085,148.922
C08067=1141.059,156.982,-59.270,-178.635,7.083,148.922
C08068=1141.065,156.732,-59.249,-178.638,7.080,148.923
C08069=1141.068,156.483,-59.227,-178.641,7.079,148.923
C08070=1141.073,156.235,-59.206,-178.644,7.077,148.924
C08071=1141.078,155.986,-59.185,-178.647,7.074,148.924
C08072=1141.082,155.736,-59.163,-178.649,7.072,148.924
C08073=1141.087,155.488,-59.141,-178.652,7.071,148.924
C08074=1141.093,155.238,-59.120,-178.655,7.068,148.925
C08075=1141.097,154.989,-59.098,-178.658,7.066,148.925
C08076=1141.101,154.740,-59.077,-178.661,7.065,148.926
C08077=1141.106,154.491,-59.056,-178.664,7.062,148.926
C08078=1141.111,154.243,-59.034,-178.666,7.060,148.926
C08079=1141.116,153.993,-59.013,-178.669,7.058,148.927
C08080=1141.120,153.744,-58.991,-178.672,7.056,148.927
C08081=1141.126,153.495,-58.970,-178.675,7.054,148.927
C08082=1141.130,153.247,-58.949,-178.678,7.052,148.928
C08083=1141.134,152.997,-58.928,-178.680,7.050,148.928
C08084=1141.139,152.748,-58.906,-178.683,7.048,148.928
C08085=1141.144,152.499,-58.885,-178.686,7.046,148.929
C08086=1141.148,152.250,-58.864,-178.689,7.044,148.929
C08087=1141.153,152.000,-58.843,-178.692,7.042,148.929
C08088=1141.158,151.752,-58.821,-178.695,7.040,148.930
C08089=1141.163,151.503,-58.800,-178.697,7.038,148.930
C08090=1141.167,151.254,-58.779,-178.700,7.036,148.930
C08091=1141.172,151.005,-58.758,-178.703,7.034,148.931
C08092=1141.177,150.755,-58.737,-178.706,7.032,148.931
C08093=1141.182,150.506,-58.715,-178.708,7.030,148.931
C08094=1141.186,150.257,-58.695,-178.712,7.028,148.932
C08095=1141.191,150.009,-58.673,-178.714,7.026,148.932
C08096=1141.196,149.759,-58.652,-178.717,7.024,148.932
C08097=1141.200,149.510,-58.631,-178.719,7.022,148.933
C08098=1141.205,149.261,-58.609,-178.723,7.020,148.933
C08099=1141.210,149.012,-58.589,-178.725,7.018,148.933
C08100=1141.215,148.763,-58.568,-178.728,7.016,148.934
C08101=1141.219,148.514,-58.546,-178.731,7.015,148.934
C08102=1141.225,148.265,-58.525,-178.734,7.012,148.934
C08103=1141.229,148.016,-58.505,-178.736,7.010,148.935
C08104=1141.234,147.766,-58.484,-178.739,7.008,148.935
C08105=1141.238,147.518,-58.463,-178.742,7.007,148.935
C08106=1141.243,147.269,-58.442,-178.745,7.004,148.936
C08107=1141.248,147.019,-58.421,-178.748,7.002,148.936
C08108=1141.253,146.770,-58.400,-178.751,7.001,148.937
C08109=1141.257,146.522,-58.379,-178.753,6.999,148.937
C08110=1141.262,146.273,-58.358,-178.756,6.996,148.937
C08111=1141.267,146.024,-58.337,-178.759,6.994,148.938
C08112=1141.271,145.774,-58.317,-178.762,6.993,148.938
C08113=1141.276,145.525,-58.296,-178.764,6.991,148.938
C08114=1141.281,145.275,-58.275,-178.768,6.989,148.939
C08115=1141.285,145.027,-58.254,-178.770,6.987,148.939
C08116=1141.291,144.778,-58.233,-178.773,6.985,148.939
C08117=1141.295,144.529,-58.212,-178.775,6.983,148.940
C08118=1141.300,144.280,-58.191,-178.779,6.981,148.940
C08119=1141.305,144.031,-58.171,-178.781,6.979,148.940
C08120=1141.310,143.781,-58.150,-178.784,6.977,148.941
C08121=1141.314,143.532,-58.130,-178.787,6.975,148.941
C08122=1141.319,143.283,-58.109,-178.790,6.973,148.942
C08123=1141.324,143.034,-58.088,-178.793,6.971,148.942
C08124=1141.328,142.785,-58.068,-178.795,6.970,148.942
C08125=1141.333,142.536,-58.047,-178.798,6.968,148.943
C08126=1141.338,142.287,-58.027,-178.801,6.966,148.943
C08127=1141.342,142.037,-58.005,-178.804,6.963,148.943
C08128=1141.347,141.788,-57.985,-178.806,6.962,148.944
C08129=1141.352,141.539,-57.964,-178.809,6.960,148.944
C08130=1141.357,141.290,-57.944,-178.812,6.958,148.944
C08131=1141.361,141.041,-57.923,-178.815,6.956,148.945
C08132=1141.366,140.792,-57.902,-178.818,6.954,148.945
C08133=1141.371,140.543,-57.882,-178.821,6.952,148.946
C08134=1141.375,140.294,-57.861,-178.823,6.950,148.946
C08135=1141.380,140.045,-57.840,-178.826,6.949,148.946
C08136=1141.385,139.796,-57.820,-178.829,6.947,148.947
C08137=1141.390,139.546,-57.799,-178.832,6.945,148.947
C08138=1141.394,139.297,-57.779,-178.835,6.943,148.948
C08139=1141.400,139.049,-57.759,-178.837,6.941,148.948
C08140=1141.405,138.799,-57.738,-178.840,6.939,148.948
C08141=1141.409,138.550,-57.718,-178.842,6.937,148.948
C08142=1141.414,138.301,-57.698,-178.845,6.936,148.949
C08143=1141.419,138.052,-57.677,-178.848,6.933,148.949
C08144=1141.423,137.803,-57.656,-178.851,6.931,148.950
C08145=1141.428,137.554,-57.637,-178.854,6.930,148.950
C08146=1141.432,137.305,-57.616,-178.857,6.928,148.950
C08147=1141.438,137.055,-57.595,-178.859,6.926,148.951
C08148=1141.442,136.806,-57.575,-178.863,6.924,148.951
C08149=1141.447,136.557,-57.555,-178.865,6.922,148.952
C08150=1141.451,136.308,-57.535,-178.868,6.920,148.952
C08151=1141.456,136.059,-57.514,-178.871,6.919,148.952
C08152=1141.461,135.810,-57.494,-178.873,6.917,148.953
C08153=1141.466,135.561,-57.474,-178.876,6.915,148.953
C08154=1141.471,135.312,-57.454,-178.880,6.913,148.954
C08155=1141.476,135.063,-57.433,-178.882,6.911,148.954
C08156=1141.481,134.813,-57.413,-178.884,6.909,148.954
C08157=1141.485,134.564,-57.393,-178.887,6.907,148.954
C08158=1141.489,134.315,-57.373,-178.890,6.906,148.955
C08159=1141.494,134.066,-57.353,-178.893,6.904,148.955
C08160=1141.499,133.816,-57.332,-178.895,6.902,148.956
C08161=1141.505,133.567,-57.313,-178.899,6.900,148.956
C08162=1141.509,133.319,-57.292,-178.901,6.898,148.956
C08163=1141.514,133.070,-57.272,-178.904,6.896,148.957
C08164=1141.518,132.820,-57.252,-178.907,6.895,148.957
C08165=1141.523,132.571,-57.232,-178.910,6.893,148.958
C08166=1141.527,132.321,-57.212,-178.912,6.891,148.958
C08167=1141.533,132.073,-57.192,-178.915,6.890,148.958
C08168=1141.538,131.804,-57.171,-178.918,6.887,148.959
C08169=1141.543,131.536,-57.150,-178.921,6.885,148.959
C08170=1141.548,131.267,-57.127,-178.924,6.884,148.960
C08171=1141.553,130.999,-57.106,-178.928,6.881,148.960
C08172=1141.558,130.750,-57.086,-178.930,6.880,148.961
C08173=1141.563,130.500,-57.065,-178.933,6.878,148.961
C08174=1141.568,130.251,-57.045,-178.935,6.876,148.961
C08175=1141.573,130.002,-57.026,-178.938,6.874,148.962
C08176=1141.578,129.752,-57.006,-178.941,6.873,148.962
C08177=1141.582,129.503,-56.986,-178.944,6.870,148.962
C08178=1141.587,129.254,-56.966,-178.947,6.868,148.963
C08179=1141.591,129.005,-56.946,-178.949,6.867,148.963
C08180=1141.597,128.756,-56.926,-178.952,6.865,148.964
C08181=1141.601,128.507,-56.907,-178.955,6.863,148.964
C08182=1141.606,128.258,-56.886,-178.958,6.862,148.964
C08183=1141.611,128.009,-56.867,-178.960,6.860,148.965
C08184=1141.616,127.759,-56.847,-178.963,6.858,148.965
C08185=1141.620,127.510,-56.827,-178.966,6.857,148.966
C08186=1141.625,127.261,-56.807,-178.968,6.855,148.966
C08187=1141.630,127.012,-56.788,-178.972,6.852,148.966
C08188=1141.635,126.763,-56.768,-178.974,6.851,148.967
C08189=1141.640,126.513,-56.748,-178.977,6.849,148.967
C08190=1141.644,126.264,-56.728,-178.980,6.847,148.967
C08191=1141.650,126.015,-56.709,-178.983,6.846,148.968
C08192=1141.653,125.766,-56.689,-178.985,6.844,148.968
C08193=1141.658,125.517,-56.670,-178.989,6.843,148.969
C08194=1141.664,125.268,-56.650,-178.991,6.841,148.969
C08195=1141.668,125.018,-56.631,-178.994,6.839,148.970
C08196=1141.673,124.769,-56.610,-178.997,6.837,148.970
C08197=1141.678,124.520,-56.591,-178.999,6.836,148.971
C08198=1141.683,124.271,-56.571,-179.002,6.834,148.971
C08199=1141.688,124.021,-56.552,-179.006,6.832,148.971
C08200=1141.693,123.772,-56.533,-179.008,6.830,148.972
C08201=1141.697,123.524,-56.513,-179.011,6.828,148.972
C08202=1141.701,123.274,-56.493,-179.014,6.826,148.972
C08203=1141.707,123.025,-56.474,-179.016,6.825,148.973
C08204=1141.711,122.776,-56.454,-179.019,6.823,148.973
C08205=1141.716,122.526,-56.434,-179.022,6.821,148.974
C08206=1141.722,122.277,-56.415,-179.025,6.820,148.974
C08207=1141.726,122.028,-56.396,-179.027,6.818,148.974
C08208=1141.730,121.778,-56.376,-179.030,6.816,148.975
C08209=1141.736,121.530,-56.357,-179.033,6.815,148.975
C08210=1141.740,121.280,-56.338,-179.035,6.813,148.976
C08211=1141.745,121.031,-56.319,-179.038,6.811,148.976
C08212=1141.750,120.782,-56.299,-179.041,6.810,148.977
C08213=1141.754,120.532,-56.280,-179.044,6.808,148.977
C08214=1141.760,120.283,-56.260,-179.046,6.806,148.977
C08215=1141.765,120.034,-56.241,-179.049,6.804,148.978
C08216=1141.769,119.785,-56.222,-179.052,6.803,148.978
C08217=1141.774,119.536,-56.202,-179.055,6.801,148.979
C08218=1141.779,119.287,-56.183,-179.057,6.799,148.979
C08219=1141.783,119.038,-56.164,-179.061,6.797,148.979
C08220=1141.788,118.788,-56.144,-179.063,6.795,148.980
C08221=1141.793,118.539,-56.125,-179.067,6.794,148.980
C08222=1141.798,118.290,-56.105,-179.069,6.792,148.981
C08223=1141.803,118.041,-56.087,-179.072,6.791,148.981
C08224=1141.807,117.791,-56.067,-179.075,6.789,148.982
C08225=1141.813,117.543,-56.048,-179.077,6.787,148.982
C08226=1141.817,117.293,-56.029,-179.080,6.785,148.982
C08227=1141.822,117.044,-56.010,-179.083,6.784,148.983
C08228=1141.827,116.794,-55.990,-179.086,6.782,148.983
C08229=1141.832,116.546,-55.972,-179.088,6.780,148.984
C08230=1141.836,116.296,-55.952,-179.091,6.779,148.984
C08231=1141.842,116.047,-55.933,-179.094,6.777,148.984
C08232=1141.846,115.798,-55.914,-179.097,6.775,148.985
C08233=1141.851,115.549,-55.895,-179.099,6.774,148.985
C08234=1141.856,115.299,-55.876,-179.102,6.772,148.986
C08235=1141.861,115.050,-55.857,-179.105,6.771,148.986
C08236=1141.866,114.801,-55.837,-179.108,6.769,148.987
C08237=1141.871,114.552,-55.819,-179.111,6.767,148.987
C08238=1141.875,114.302,-55.799,-179.113,6.766,148.987
C08239=1141.880,114.054,-55.781,-179.116,6.764,148.988
C08240=1141.885,113.804,-55.761,-179.119,6.762,148.988
C08241=1141.890,113.555,-55.743,-179.122,6.760,148.989
C08242=1141.894,113.305,-55.723,-179.124,6.759,148.989
C08243=1141.900,113.056,-55.704,-179.127,6.757,148.989
C08244=1141.905,112.807,-55.686,-179.130,6.755,148.990
C08245=1141.909,112.558,-55.666,-179.132,6.754,148.990
C08246=1141.914,112.309,-55.648,-179.135,6.752,148.991
C08247=1141.919,112.059,-55.629,-179.138,6.751,148.991
C08248=1141.924,111.810,-55.610,-179.141,6.749,148.992
C08249=1141.928,111.561,-55.590,-179.144,6.747,148.992
C08250=1141.933,111.312,-55.573,-179.147,6.746,148.993
C08251=1141.939,111.063,-55.553,-179.149,6.744,148.993
C08252=1141.943,110.813,-55.535,-179.151,6.743,148.993
C08253=1141.948,110.564,-55.516,-179.154,6.741,148.994
C08254=1141.952,110.314,-55.497,-179.157,6.740,148.994
C08255=1141.958,110.065,-55.478,-179.160,6.738,148.995
C08256=1141.962,109.817,-55.459,-179.162,6.736,148.995
C08257=1141.967,109.567,-55.441,-179.166,6.735,148.996
C08258=1141.972,109.318,-55.422,-179.168,6.733,148.996
C08259=1141.977,109.069,-55.404,-179.171,6.732,148.996
C08260=1141.982,108.819,-55.384,-179.174,6.730,148.997
C08261=1141.987,108.570,-55.366,-179.176,6.728,148.997
C08262=1141.991,108.321,-55.347,-179.179,6.727,148.998
C08263=1141.996,108.071,-55.328,-179.182,6.725,148.998
C08264=1142.001,107.822,-55.310,-179.185,6.723,148.999
C08265=1142.006,107.573,-55.291,-179.188,6.722,148.999
C08266=1142.011,107.323,-55.273,-179.191,6.720,149.000
C08267=1142.015,107.075,-55.254,-179.193,6.719,149.000
C08268=1142.021,106.825,-55.235,-179.196,6.717,149.000
C08269=1142.025,106.576,-55.216,-179.199,6.715,149.001
C08270=1142.030,106.327,-55.198,-179.202,6.714,149.001
C08271=1142.035,106.077,-55.179,-179.204,6.713,149.002
C08272=1142.040,105.809,-55.159,-179.207,6.711,149.002
C08273=1142.046,105.541,-55.139,-179.210,6.709,149.003
C08274=1142.051,105.272,-55.120,-179.213,6.707,149.003
C08275=1142.057,105.004,-55.100,-179.216,6.705,149.003
C08276=1142.061,104.754,-55.081,-179.219,6.704,149.004
C08277=1142.066,104.505,-55.063,-179.222,6.702,149.005
C08278=1142.070,104.256,-55.045,-179.224,6.701,149.005
C08279=1142.076,104.007,-55.026,-179.227,6.699,149.005
C08280=1142.080,103.757,-55.007,-179.230,6.697,149.006
C08281=1142.085,103.508,-54.989,-179.233,6.696,149.006
C08282=1142.090,103.259,-54.971,-179.235,6.694,149.007
C08283=1142.095,103.009,-54.952,-179.238,6.694,149.007
C08284=1142.100,102.760,-54.934,-179.241,6.692,149.008
C08285=1142.104,102.511,-54.916,-179.243,6.690,149.008
C08286=1142.109,102.262,-54.898,-179.246,6.689,149.008
C08287=1142.115,102.012,-54.879,-179.249,6.687,149.009
C08288=1142.119,101.763,-54.860,-179.252,6.685,149.009
C08289=1142.124,101.514,-54.842,-179.254,6.683,149.010
C08290=1142.129,101.265,-54.824,-179.258,6.682,149.010
C08291=1142.134,101.016,-54.806,-179.260,6.680,149.011
C08292=1142.138,100.766,-54.788,-179.262,6.680,149.011
C08293=1142.144,100.516,-54.769,-179.265,6.678,149.012
C08294=1142.148,100.268,-54.751,-179.268,6.676,149.012
C08295=1142.153,100.019,-54.733,-179.271,6.675,149.012
C08296=1142.158,99.769,-54.715,-179.274,6.673,149.013
C08297=1142.162,99.519,-54.696,-179.277,6.672,149.013
C08298=1142.167,99.270,-54.678,-179.279,6.670,149.014
C08299=1142.172,99.021,-54.660,-179.282,6.668,149.014
C08300=1142.178,98.772,-54.642,-179.285,6.667,149.015
C08301=1142.183,98.522,-54.624,-179.287,6.666,149.015
C08302=1142.188,98.273,-54.606,-179.290,6.664,149.016
C08303=1142.192,98.023,-54.587,-179.293,6.663,149.016
C08304=1142.197,97.774,-54.569,-179.296,6.661,149.017
C08305=1142.202,97.525,-54.551,-179.298,6.659,149.017
C08306=1142.207,97.276,-54.533,-179.301,6.658,149.017
C08307=1142.212,97.027,-54.515,-179.304,6.656,149.018
C08308=1142.217,96.778,-54.498,-179.306,6.655,149.019
C08309=1142.222,96.528,-54.480,-179.309,6.654,149.019
C08310=1142.226,96.279,-54.462,-179.312,6.652,149.019
C08311=1142.231,96.029,-54.443,-179.315,6.650,149.020
C08312=1142.236,95.780,-54.425,-179.317,6.649,149.020
C08313=1142.241,95.531,-54.407,-179.320,6.647,149.021
C08314=1142.246,95.282,-54.389,-179.323,6.646,149.021
C08315=1142.250,95.033,-54.371,-179.325,6.645,149.022
C08316=1142.255,94.783,-54.353,-179.328,6.643,149.022
C08317=1142.261,94.534,-54.336,-179.331,6.642,149.023
C08318=1142.265,94.284,-54.318,-179.334,6.640,149.023
C08319=1142.270,94.035,-54.300,-179.337,6.639,149.024
C08320=1142.275,93.786,-54.282,-179.340,6.637,149.024
C08321=1142.280,93.536,-54.264,-179.342,6.635,149.024
C08322=1142.285,93.287,-54.246,-179.344,6.634,149.025
C08323=1142.289,93.038,-54.228,-179.347,6.633,149.025
C08324=1142.295,92.788,-54.211,-179.350,6.631,149.026
C08325=1142.300,92.539,-54.193,-179.353,6.630,149.026
C08326=1142.304,92.290,-54.175,-179.356,6.628,149.027
C08327=1142.309,92.041,-54.157,-179.358,6.627,149.027
C08328=1142.315,91.791,-54.139,-179.361,6.626,149.028
C08329=1142.320,91.542,-54.121,-179.364,6.624,149.028
C08330=1142.324,91.292,-54.103,-179.367,6.623,149.029
C08331=1142.329,91.044,-54.086,-179.369,6.621,149.029
C08332=1142.334,90.794,-54.069,-179.372,6.619,149.029
C08333=1142.339,90.545,-54.051,-179.374,6.618,149.030
C08334=1142.344,90.295,-54.033,-179.378,6.617,149.031
C08335=1142.349,90.046,-54.015,-179.380,6.615,149.031
C08336=1142.354,89.796,-53.998,-179.383,6.614,149.031
C08337=1142.359,89.547,-53.980,-179.386,6.612,149.032
C08338=1142.363,89.298,-53.963,-179.388,6.611,149.032
C08339=1142.368,89.049,-53.945,-179.391,6.610,149.033
C08340=1142.373,88.799,-53.927,-179.394,6.608,149.033
C08341=1142.378,88.550,-53.910,-179.397,6.607,149.034
C08342=1142.383,88.300,-53.892,-179.399,6.605,149.034
C08343=1142.388,88.051,-53.874,-179.402,6.604,149.035
C08344=1142.393,87.802,-53.857,-179.405,6.603,149.035
C08345=1142.397,87.553,-53.839,-179.407,6.601,149.036
C08346=1142.403,87.303,-53.822,-179.410,6.599,149.036
C08347=1142.408,87.054,-53.804,-179.413,6.598,149.037
C08348=1142.412,86.804,-53.787,-179.416,6.597,149.037
C08349=1142.417,86.555,-53.769,-179.418,6.595,149.038
C08350=1142.422,86.307,-53.752,-179.421,6.594,149.038
C08351=1142.428,86.057,-53.734,-179.424,6.592,149.038
C08352=1142.432,85.808,-53.717,-179.427,6.590,149.039
C08353=1142.437,85.558,-53.700,-179.429,6.590,149.040
C08354=1142.442,85.309,-53.682,-179.432,6.588,149.040
C08355=1142.447,85.059,-53.664,-179.435,6.587,149.040
C08356=1142.451,84.810,-53.647,-179.437,6.585,149.041
C08357=1142.457,84.560,-53.630,-179.440,6.584,149.041
C08358=1142.462,84.311,-53.612,-179.443,6.583,149.042
C08359=1142.466,84.062,-53.595,-179.445,6.581,149.042
C08360=1142.471,83.812,-53.578,-179.448,6.579,149.043
C08361=1142.477,83.563,-53.560,-179.451,6.579,149.043
C08362=1142.481,83.314,-53.544,-179.454,6.577,149.044
C08363=1142.486,83.065,-53.526,-179.456,6.576,149.044
C08364=1142.491,82.815,-53.508,-179.459,6.574,149.045
C08365=1142.496,82.566,-53.492,-179.462,6.574,149.045
C08366=1142.501,82.316,-53.474,-179.464,6.572,149.046
C08367=1142.506,82.067,-53.456,-179.467,6.570,149.046
C08368=1142.511,81.818,-53.440,-179.470,6.569,149.047
C08369=1142.516,81.569,-53.422,-179.473,6.568,149.047
C08370=1142.520,81.319,-53.405,-179.475,6.566,149.048
C08371=1142.526,81.069,-53.388,-179.478,6.565,149.048
C08372=1142.531,80.820,-53.370,-179.481,6.563,149.048
C08373=1142.535,80.571,-53.353,-179.483,6.562,149.049
C08374=1142.541,80.322,-53.337,-179.486,6.561,149.050
C08375=1142.545,80.072,-53.320,-179.489,6.559,149.050
C08376=1142.550,79.804,-53.301,-179.492,6.558,149.050
C08377=1142.556,79.536,-53.282,-179.495,6.556,149.051
C08378=1142.561,79.267,-53.264,-179.498,6.555,149.051
C08379=1142.566,78.998,-53.245,-179.501,6.553,149.052
C08380=1142.571,78.749,-53.229,-179.503,6.552,149.053
C08381=1142.577,78.500,-53.212,-179.506,6.551,149.053
C08382=1142.581,78.251,-53.194,-179.508,6.549,149.053
C08383=1142.586,78.001,-53.177,-179.512,6.548,149.054
C08384=1142.591,77.752,-53.161,-179.514,6.547,149.055
C08385=1142.596,77.502,-53.144,-179.517,6.545,149.055
C08386=1142.601,77.253,-53.127,-179.520,6.544,149.056
C08387=1142.606,77.003,-53.110,-179.522,6.543,149.056
C08388=1142.610,76.754,-53.092,-179.525,6.541,149.056
C08389=1142.616,76.505,-53.075,-179.527,6.540,149.057
C08390=1142.621,76.256,-53.059,-179.531,6.539,149.058
C08391=1142.626,76.006,-53.041,-179.533,6.538,149.058
C08392=1142.630,75.756,-53.025,-179.536,6.536,149.058
C08393=1142.636,75.507,-53.008,-179.538,6.534,149.059
C08394=1142.641,75.258,-52.991,-179.541,6.534,149.059
C08395=1142.646,75.008,-52.974,-179.544,6.532,149.060
C08396=1142.650,74.759,-52.957,-179.546,6.531,149.060
C08397=1142.655,74.510,-52.941,-179.549,6.530,149.061
C08398=1142.661,74.260,-52.924,-179.552,6.528,149.061
C08399=1142.665,74.011,-52.907,-179.555,6.527,149.062
C08400=1142.671,73.761,-52.890,-179.557,6.525,149.062
C08401=1142.675,73.512,-52.873,-179.560,6.525,149.063
C08402=1142.680,73.262,-52.857,-179.563,6.523,149.063
C08403=1142.686,73.013,-52.840,-179.565,6.521,149.064
C08404=1142.690,72.764,-52.823,-179.568,6.520,149.064
C08405=1142.695,72.514,-52.807,-179.571,6.519,149.065
C08406=1142.700,72.265,-52.790,-179.574,6.517,149.065
C08407=1142.705,72.016,-52.773,-179.576,6.517,149.066
C08408=1142.709,71.766,-52.756,-179.579,6.515,149.066
C08409=1142.715,71.517,-52.739,-179.582,6.514,149.067
C08410=1142.720,71.268,-52.723,-179.584,6.513,149.067
C08411=1142.724,71.018,-52.706,-179.587,6.511,149.068
C08412=1142.730,70.769,-52.689,-179.590,6.510,149.068
C08413=1142.734,70.520,-52.673,-179.592,6.509,149.069
C08414=1142.739,70.270,-52.657,-179.595,6.507,149.069
C08415=1142.745,70.020,-52.640,-179.598,6.506,149.070
C08416=1142.750,69.771,-52.623,-179.600,6.505,149.070
C08417=1142.755,69.522,-52.607,-179.603,6.504,149.071
C08418=1142.759,69.273,-52.590,-179.606,6.502,149.071
C08419=1142.764,69.023,-52.573,-179.608,6.501,149.072
C08420=1142.769,68.774,-52.556,-179.611,6.500,149.072
C08421=1142.774,68.524,-52.541,-179.614,6.498,149.073
C08422=1142.779,68.275,-52.524,-179.616,6.498,149.073
C08423=1142.784,68.025,-52.507,-179.619,6.496,149.074
C08424=1142.789,67.776,-52.490,-179.622,6.494,149.074
C08425=1142.794,67.527,-52.475,-179.624,6.493,149.075
C08426=1142.799,67.277,-52.458,-179.627,6.492,149.075
C08427=1142.805,67.028,-52.441,-179.629,6.491,149.076
C08428=1142.809,66.779,-52.424,-179.632,6.490,149.076
C08429=1142.814,66.528,-52.409,-179.635,6.488,149.077
C08430=1142.819,66.280,-52.392,-179.637,6.488,149.077
C08431=1142.823,66.030,-52.376,-179.640,6.486,149.078
C08432=1142.829,65.781,-52.360,-179.643,6.485,149.078
C08433=1142.834,65.531,-52.343,-179.646,6.484,149.079
C08434=1142.839,65.282,-52.326,-179.648,6.482,149.079
C08435=1142.844,65.033,-52.310,-179.651,6.481,149.080
C08436=1142.849,64.783,-52.294,-179.654,6.480,149.080
C08437=1142.854,64.534,-52.277,-179.656,6.478,149.081
C08438=1142.858,64.284,-52.262,-179.659,6.477,149.081
C08439=1142.863,64.035,-52.245,-179.662,6.476,149.082
C08440=1142.868,63.785,-52.229,-179.665,6.475,149.082
C08441=1142.874,63.536,-52.212,-179.667,6.474,149.083
C08442=1142.878,63.286,-52.196,-179.670,6.472,149.083
C08443=1142.884,63.037,-52.180,-179.672,6.472,149.084
C08444=1142.888,62.787,-52.163,-179.675,6.470,149.084
C08445=1142.893,62.539,-52.147,-179.678,6.469,149.085
C08446=1142.898,62.288,-52.131,-179.680,6.468,149.085
C08447=1142.903,62.040,-52.115,-179.683,6.466,149.086
C08448=1142.908,61.790,-52.099,-179.686,6.466,149.087
C08449=1142.913,61.541,-52.083,-179.688,6.464,149.087
C08450=1142.919,61.291,-52.067,-179.691,6.462,149.087
C08451=1142.923,61.042,-52.050,-179.693,6.461,149.088
C08452=1142.928,60.793,-52.035,-179.697,6.460,149.089
C08453=1142.933,60.543,-52.018,-179.699,6.459,149.089
C08454=1142.938,60.294,-52.003,-179.701,6.458,149.089
C08455=1142.943,60.044,-51.986,-179.705,6.456,149.090
C08456=1142.948,59.795,-51.970,-179.707,6.456,149.090
C08457=1142.953,59.545,-51.954,-179.710,6.454,149.091
C08458=1142.958,59.296,-51.938,-179.712,6.453,149.092
C08459=1142.963,59.046,-51.922,-179.715,6.452,149.092
C08460=1142.968,58.797,-51.906,-179.718,6.450,149.092
C08461=1142.973,58.548,-51.890,-179.720,6.450,149.093
C08462=1142.978,58.298,-51.873,-179.723,6.448,149.094
C08463=1142.983,58.049,-51.858,-179.725,6.447,149.094
C08464=1142.988,57.799,-51.842,-179.729,6.446,149.095
C08465=1142.993,57.550,-51.826,-179.731,6.445,149.095
C08466=1142.998,57.300,-51.810,-179.733,6.443,149.096
C08467=1143.003,57.050,-51.794,-179.737,6.442,149.096
C08468=1143.008,56.801,-51.778,-179.739,6.441,149.097
C08469=1143.014,56.552,-51.762,-179.742,6.440,149.097
C08470=1143.018,56.302,-51.746,-179.744,6.439,149.098
C08471=1143.024,56.053,-51.730,-179.747,6.437,149.098
C08472=1143.028,55.803,-51.714,-179.749,6.437,149.099
C08473=1143.033,55.554,-51.699,-179.752,6.435,149.099
C08474=1143.038,55.305,-51.683,-179.755,6.434,149.100
C08475=1143.043,55.055,-51.667,-179.757,6.433,149.100
C08476=1143.048,54.806,-51.651,-179.761,6.432,149.101
C08477=1143.054,54.556,-51.636,-179.763,6.431,149.101
C08478=1143.058,54.307,-51.619,-179.765,6.429,149.102
C08479=1143.063,54.057,-51.603,-179.768,6.429,149.102
C08480=1143.069,53.789,-51.586,-179.771,6.427,149.103
C08481=1143.074,53.521,-51.570,-179.774,6.426,149.104
C08482=1143.079,53.252,-51.552,-179.776,6.425,149.104
C08483=1143.085,52.982,-51.536,-179.779,6.424,149.105
C08484=1143.090,52.734,-51.520,-179.782,6.422,149.105
C08485=1143.095,52.484,-51.504,-179.785,6.422,149.106
C08486=1143.100,52.234,-51.488,-179.788,6.420,149.106
C08487=1143.105,51.985,-51.473,-179.790,6.419,149.107
C08488=1143.110,51.736,-51.458,-179.793,6.418,149.107
C08489=1143.115,51.486,-51.442,-179.795,6.417,149.108
C08490=1143.120,51.236,-51.426,-179.798,6.415,149.108
C08491=1143.125,50.987,-51.410,-179.801,6.415,149.109
C08492=1143.130,50.738,-51.395,-179.803,6.413,149.109
C08493=1143.135,50.488,-51.379,-179.806,6.412,149.110
C08494=1143.140,50.239,-51.363,-179.809,6.411,149.110
C08495=1143.145,49.990,-51.348,-179.811,6.409,149.111
C08496=1143.150,49.740,-51.333,-179.814,6.409,149.111
C08497=1143.155,49.490,-51.317,-179.817,6.407,149.112
C08498=1143.160,49.241,-51.301,-179.819,6.406,149.112
C08499=1143.165,48.992,-51.286,-179.822,6.405,149.113
C08500=1143.170,48.742,-51.271,-179.824,6.404,149.114
C08501=1143.175,48.492,-51.255,-179.827,6.403,149.114
C08502=1143.180,48.243,-51.240,-179.829,6.402,149.114
C08503=1143.185,47.994,-51.224,-179.833,6.401,149.115
C08504=1143.190,47.744,-51.209,-179.835,6.400,149.116
C08505=1143.195,47.495,-51.193,-179.838,6.398,149.116
C08506=1143.200,47.245,-51.178,-179.840,6.398,149.117
C08507=1143.205,46.996,-51.162,-179.843,6.396,149.117
C08508=1143.210,46.747,-51.147,-179.845,6.396,149.118
C08509=1143.215,46.497,-51.131,-179.848,6.394,149.118
C08510=1143.220,46.247,-51.115,-179.850,6.393,149.119
C08511=1143.225,45.998,-51.100,-179.854,6.392,149.119
C08512=1143.230,45.749,-51.085,-179.856,6.391,149.120
C08513=1143.236,45.499,-51.069,-179.859,6.389,149.120
C08514=1143.240,45.250,-51.055,-179.861,6.389,149.121
C08515=1143.245,44.999,-51.039,-179.864,6.387,149.121
C08516=1143.250,44.750,-51.024,-179.866,6.386,149.122
C08517=1143.255,44.501,-51.009,-179.869,6.386,149.122
C08518=1143.261,44.252,-50.993,-179.872,6.384,149.123
C08519=1143.265,44.002,-50.978,-179.874,6.384,149.124
C08520=1143.271,43.753,-50.962,-179.877,6.382,149.124
C08521=1143.275,43.503,-50.948,-179.879,6.381,149.124
C08522=1143.280,43.253,-50.932,-179.882,6.380,149.125
C08523=1143.285,43.004,-50.917,-179.884,6.379,149.126
C08524=1143.291,42.755,-50.902,-179.887,6.378,149.126
C08525=1143.295,42.506,-50.887,-179.890,6.377,149.127
C08526=1143.301,42.256,-50.872,-179.893,6.375,149.127
C08527=1143.305,42.007,-50.857,-179.895,6.375,149.128
C08528=1143.310,41.756,-50.841,-179.898,6.373,149.128
C08529=1143.316,41.507,-50.825,-179.900,6.373,149.129
C08530=1143.321,41.257,-50.811,-179.903,6.371,149.129
C08531=1143.326,41.008,-50.795,-179.906,6.370,149.130
C08532=1143.331,40.759,-50.780,-179.908,6.370,149.130
C08533=1143.335,40.510,-50.765,-179.911,6.368,149.131
C08534=1143.341,40.260,-50.750,-179.913,6.368,149.131
C08535=1143.346,40.011,-50.735,-179.916,6.366,149.132
C08536=1143.351,39.761,-50.720,-179.919,6.365,149.133
C08537=1143.356,39.512,-50.706,-179.921,6.364,149.133
C08538=1143.361,39.262,-50.690,-179.924,6.363,149.134
C08539=1143.365,39.012,-50.675,-179.927,6.362,149.134
C08540=1143.371,38.762,-50.660,-179.929,6.361,149.135
C08541=1143.376,38.513,-50.645,-179.932,6.360,149.135
C08542=1143.381,38.263,-50.630,-179.934,6.359,149.136
C08543=1143.386,38.014,-50.615,-179.937,6.358,149.136
C08544=1143.391,37.765,-50.600,-179.940,6.357,149.137
C08545=1143.396,37.515,-50.585,-179.942,6.356,149.137
C08546=1143.401,37.266,-50.570,-179.945,6.355,149.138
C08547=1143.407,37.016,-50.555,-179.947,6.354,149.138
C08548=1143.411,36.767,-50.540,-179.950,6.352,149.139
C08549=1143.416,36.518,-50.525,-179.953,6.352,149.139
C08550=1143.422,36.268,-50.510,-179.955,6.351,149.140
C08551=1143.426,36.019,-50.495,-179.958,6.350,149.141
C08552=1143.432,35.769,-50.480,-179.960,6.349,149.141
C08553=1143.437,35.519,-50.465,-179.963,6.347,149.142
C08554=1143.442,35.270,-50.451,-179.966,6.347,149.142
C08555=1143.447,35.020,-50.436,-179.968,6.346,149.143
C08556=1143.452,34.771,-50.421,-179.971,6.344,149.143
C08557=1143.457,34.522,-50.406,-179.973,6.344,149.144
C08558=1143.462,34.272,-50.391,-179.976,6.342,149.144
C08559=1143.467,34.022,-50.376,-179.979,6.342,149.145
C08560=1143.472,33.773,-50.362,-179.981,6.341,149.145
C08561=1143.478,33.523,-50.347,-179.984,6.339,149.146
C08562=1143.482,33.274,-50.332,-179.986,6.339,149.146
C08563=1143.487,33.024,-50.318,-179.989,6.337,149.147
C08564=1143.492,32.775,-50.303,-179.992,6.337,149.148
C08565=1143.498,32.525,-50.288,-179.994,6.336,149.148
C08566=1143.502,32.276,-50.273,-179.997,6.334,149.148
C08567=1143.507,32.026,-50.259,-179.999,6.334,149.149
C08568=1143.512,31.776,-50.245,179.998,6.332,149.150
C08569=1143.518,31.527,-50.229,179.996,6.331,149.150
C08570=1143.523,31.278,-50.215,179.993,6.331,149.151
C08571=1143.528,31.028,-50.201,179.990,6.329,149.151
C08572=1143.533,30.779,-50.186,179.988,6.329,149.152
C08573=1143.538,30.529,-50.171,179.985,6.327,149.152
C08574=1143.543,30.279,-50.157,179.983,6.326,149.153
C08575=1143.548,30.030,-50.142,179.980,6.326,149.153
C08576=1143.553,29.781,-50.127,179.977,6.324,149.154
C08577=1143.558,29.531,-50.113,179.975,6.324,149.155
C08578=1143.563,29.281,-50.098,179.973,6.323,149.155
C08579=1143.568,29.032,-50.083,179.970,6.321,149.155
C08580=1143.573,28.782,-50.069,179.967,6.321,149.156
C08581=1143.578,28.532,-50.055,179.964,6.319,149.157
C08582=1143.583,28.284,-50.040,179.962,6.319,149.157
C08583=1143.589,28.034,-50.025,179.960,6.318,149.158
C08584=1143.594,27.765,-50.009,179.956,6.317,149.158
C08585=1143.600,27.496,-49.995,179.954,6.316,149.159
C08586=1143.605,27.227,-49.979,179.951,6.315,149.160
C08587=1143.611,26.958,-49.962,179.948,6.313,149.160
C08588=1143.616,26.708,-49.948,179.946,6.313,149.161
C08589=1143.621,26.458,-49.934,179.943,6.312,149.161
C08590=1143.626,26.209,-49.920,179.940,6.310,149.162
C08591=1143.631,25.960,-49.906,179.938,6.310,149.162
C08592=1143.636,25.711,-49.891,179.936,6.309,149.163
C08593=1143.641,25.461,-49.876,179.933,6.308,149.163
C08594=1143.646,25.211,-49.862,179.930,6.307,149.164
C08595=1143.651,24.961,-49.848,179.928,6.306,149.165
C08596=1143.656,24.712,-49.834,179.925,6.305,149.165
C08597=1143.662,24.462,-49.819,179.923,6.304,149.165
C08598=1143.667,24.213,-49.805,179.920,6.303,149.166
C08599=1143.672,23.963,-49.791,179.917,6.302,149.167
C08600=1143.677,23.713,-49.776,179.915,6.301,149.167
C08601=1143.682,23.465,-49.762,179.913,6.300,149.168
C08602=1143.687,23.215,-49.747,179.910,6.299,149.168
C08603=1143.692,22.965,-49.733,179.907,6.298,149.169
C08604=1143.697,22.716,-49.719,179.905,6.298,149.169
C08605=1143.702,22.466,-49.705,179.902,6.296,149.170
C08606=1143.707,22.217,-49.691,179.900,6.295,149.170
C08607=1143.712,21.967,-49.676,179.897,6.295,149.171
C08608=1143.717,21.718,-49.662,179.894,6.293,149.172
C08609=1143.722,21.468,-49.648,179.892,6.293,149.172
C08610=1143.728,21.219,-49.634,179.889,6.292,149.173
C08611=1143.733,20.969,-49.620,179.887,6.291,149.173
C08612=1143.738,20.719,-49.605,179.884,6.290,149.174
C08613=1143.743,20.470,-49.591,179.882,6.289,149.174
C08614=1143.748,20.221,-49.577,179.879,6.288,149.175
C08615=1143.753,19.971,-49.563,179.876,6.287,149.175
C08616=1143.758,19.721,-49.549,179.874,6.286,149.176
C08617=1143.763,19.471,-49.535,179.872,6.286,149.176
C08618=1143.768,19.222,-49.522,179.869,6.284,149.177
C08619=1143.773,18.973,-49.507,179.867,6.283,149.178
C08620=1143.778,18.723,-49.493,179.864,6.283,149.178
C08621=1143.783,18.473,-49.479,179.861,6.281,149.179
C08622=1143.789,18.224,-49.465,179.859,6.281,149.179
C08623=1143.794,17.974,-49.451,179.856,6.280,149.180
C08624=1143.799,17.725,-49.436,179.854,6.279,149.180
C08625=1143.804,17.476,-49.423,179.851,6.278,149.181
C08626=1143.809,17.225,-49.409,179.849,6.277,149.181
C08627=1143.814,16.976,-49.395,179.847,6.276,149.182
C08628=1143.819,16.726,-49.381,179.843,6.275,149.183
C08629=1143.824,16.477,-49.367,179.841,6.274,149.183
C08630=1143.829,16.228,-49.353,179.839,6.274,149.184
C08631=1143.834,15.978,-49.339,179.836,6.272,149.184
C08632=1143.840,15.728,-49.325,179.833,6.272,149.185
C08633=1143.845,15.478,-49.311,179.831,6.271,149.185
C08634=1143.850,15.229,-49.297,179.829,6.270,149.186
C08635=1143.855,14.980,-49.283,179.826,6.269,149.186
C08636=1143.860,14.730,-49.270,179.823,6.268,149.187
C08637=1143.865,14.480,-49.256,179.821,6.268,149.188
C08638=1143.870,14.231,-49.242,179.818,6.266,149.188
C08639=1143.875,13.981,-49.227,179.816,6.265,149.189
C08640=1143.880,13.732,-49.215,179.813,6.265,149.189
C08641=1143.885,13.482,-49.201,179.811,6.264,149.190
C08642=1143.890,13.233,-49.186,179.808,6.263,149.190
C08643=1143.896,12.983,-49.173,179.806,6.262,149.191
C08644=1143.901,12.733,-49.159,179.803,6.261,149.191
C08645=1143.905,12.484,-49.145,179.801,6.261,149.192
C08646=1143.911,12.235,-49.131,179.798,6.259,149.192
C08647=1143.916,11.984,-49.118,179.795,6.259,149.193
C08648=1143.922,11.735,-49.104,179.793,6.258,149.194
C08649=1143.926,11.485,-49.091,179.790,6.257,149.194
C08650=1143.931,11.236,-49.077,179.788,6.256,149.195
C08651=1143.937,10.987,-49.063,179.786,6.255,149.195
C08652=1143.941,10.737,-49.050,179.783,6.255,149.196
C08653=1143.947,10.488,-49.036,179.781,6.254,149.196
C08654=1143.952,10.238,-49.021,179.777,6.253,149.197
C08655=1143.957,9.988,-49.008,179.775,6.252,149.197
C08656=1143.962,9.739,-48.995,179.773,6.251,149.198
C08657=1143.967,9.489,-48.981,179.770,6.250,149.199
C08658=1143.973,9.240,-48.967,179.768,6.249,149.199
C08659=1143.977,8.990,-48.954,179.765,6.248,149.200
C08660=1143.983,8.741,-48.940,179.763,6.248,149.200
C08661=1143.988,8.490,-48.927,179.761,6.247,149.201
C08662=1143.993,8.242,-48.913,179.757,6.246,149.201
C08663=1143.998,7.992,-48.899,179.755,6.245,149.202
C08664=1144.003,7.742,-48.886,179.753,6.244,149.202
C08665=1144.008,7.493,-48.872,179.750,6.243,149.203
C08666=1144.013,7.243,-48.859,179.747,6.242,149.204
C08667=1144.019,6.994,-48.845,179.745,6.241,149.204
C08668=1144.023,6.743,-48.832,179.743,6.241,149.205
C08669=1144.029,6.494,-48.819,179.740,6.240,149.205
C08670=1144.033,6.244,-48.805,179.738,6.239,149.206
C08671=1144.039,5.995,-48.792,179.735,6.238,149.206
C08672=1144.044,5.745,-48.777,179.733,6.237,149.207
C08673=1144.049,5.496,-48.765,179.730,6.236,149.207
C08674=1144.054,5.246,-48.751,179.728,6.236,149.208
C08675=1144.059,4.997,-48.738,179.725,6.234,149.208
C08676=1144.064,4.747,-48.724,179.722,6.234,149.209
C08677=1144.069,4.498,-48.711,179.720,6.233,149.210
C08678=1144.075,4.247,-48.697,179.718,6.233,149.210
C08679=1144.080,3.998,-48.684,179.715,6.232,149.211
C08680=1144.085,3.748,-48.671,179.713,6.230,149.211
C08681=1144.091,3.499,-48.657,179.710,6.230,149.212
C08682=1144.095,3.249,-48.644,179.708,6.229,149.212
C08683=1144.101,3.000,-48.631,179.705,6.229,149.213
C08684=1144.106,2.750,-48.618,179.703,6.228,149.214
C08685=1144.111,2.501,-48.604,179.700,6.227,149.214
C08686=1144.116,2.251,-48.591,179.697,6.226,149.215
C08687=1144.121,2.001,-48.577,179.695,6.225,149.215
C08688=1144.127,1.732,-48.563,179.693,6.225,149.216
C08689=1144.132,1.463,-48.549,179.689,6.223,149.217
C08690=1144.138,1.193,-48.534,179.687,6.223,149.217
C08691=1144.143,0.923,-48.520,179.685,6.222,149.218
C08692=1144.148,0.674,-48.507,179.682,6.220,149.218
C08693=1144.154,0.425,-48.493,179.679,6.220,149.219
C08694=1144.159,0.175,-48.480,179.677,6.219,149.219
C08695=1144.164,-0.074,-48.468,179.675,6.218,149.220
C08696=1144.169,-0.324,-48.454,179.672,6.218,149.220
C08697=1144.174,-0.574,-48.441,179.669,6.216,149.221
C08698=1144.180,-0.823,-48.428,179.667,6.216,149.222
C08699=1144.184,-1.073,-48.415,179.665,6.215,149.222
C08700=1144.190,-1.323,-48.402,179.662,6.215,149.223
C08701=1144.194,-1.572,-48.388,179.660,6.214,149.223
C08702=1144.199,-1.822,-48.375,179.657,6.213,149.224
C08703=1144.205,-2.071,-48.362,179.654,6.212,149.224
C08704=1144.210,-2.321,-48.349,179.652,6.211,149.225
C08705=1144.216,-2.571,-48.336,179.649,6.211,149.226
C08706=1144.220,-2.821,-48.323,179.647,6.210,149.226
C08707=1144.225,-3.070,-48.310,179.645,6.209,149.226
C08708=1144.231,-3.319,-48.296,179.642,6.209,149.227
C08709=1144.235,-3.569,-48.284,179.640,6.207,149.228
C08710=1144.241,-3.819,-48.270,179.637,6.207,149.228
C08711=1144.246,-4.068,-48.258,179.635,6.206,149.229
C08712=1144.251,-4.318,-48.245,179.632,6.205,149.229
C08713=1144.257,-4.568,-48.232,179.630,6.205,149.230
C08714=1144.262,-4.817,-48.219,179.628,6.204,149.230
C08715=1144.266,-5.067,-48.206,179.625,6.203,149.231
C08716=1144.272,-5.317,-48.193,179.622,6.202,149.232
C08717=1144.277,-5.566,-48.180,179.620,6.201,149.232
C08718=1144.282,-5.816,-48.167,179.618,6.200,149.233
C08719=1144.288,-6.066,-48.154,179.615,6.200,149.233
C08720=1144.293,-6.315,-48.141,179.613,6.199,149.234
C08721=1144.297,-6.564,-48.128,179.610,6.198,149.234
C08722=1144.303,-6.814,-48.115,179.608,6.198,149.235
C08723=1144.308,-7.063,-48.102,179.605,6.196,149.236
C08724=1144.313,-7.313,-48.089,179.602,6.196,149.236
C08725=1144.318,-7.563,-48.077,179.600,6.195,149.237
C08726=1144.324,-7.813,-48.064,179.598,6.194,149.237
C08727=1144.329,-8.062,-48.051,179.595,6.194,149.238
C08728=1144.334,-8.312,-48.038,179.593,6.193,149.238
C08729=1144.339,-8.562,-48.026,179.591,6.193,149.239
C08730=1144.344,-8.811,-48.013,179.588,6.192,149.239
C08731=1144.350,-9.061,-48.000,179.585,6.191,149.240
C08732=1144.354,-9.311,-47.987,179.583,6.190,149.241
C08733=1144.359,-9.560,-47.974,179.581,6.189,149.241
C08734=1144.365,-9.809,-47.961,179.578,6.189,149.242
C08735=1144.370,-10.059,-47.949,179.576,6.188,149.242
C08736=1144.375,-10.309,-47.936,179.573,6.187,149.243
C08737=1144.380,-10.558,-47.923,179.571,6.187,149.243
C08738=1144.385,-10.807,-47.910,179.569,6.186,149.244
C08739=1144.390,-11.057,-47.899,179.566,6.185,149.245
C08740=1144.396,-11.308,-47.885,179.563,6.184,149.245
C08741=1144.401,-11.557,-47.872,179.561,6.183,149.246
C08742=1144.406,-11.806,-47.860,179.559,6.183,149.246
C08743=1144.411,-12.056,-47.847,179.556,6.182,149.247
C08744=1144.416,-12.306,-47.834,179.554,6.181,149.247
C08745=1144.422,-12.556,-47.822,179.552,6.181,149.248
C08746=1144.427,-12.805,-47.809,179.549,6.180,149.249
C08747=1144.432,-13.055,-47.797,179.547,6.179,149.249
C08748=1144.437,-13.304,-47.784,179.544,6.179,149.250
C08749=1144.442,-13.554,-47.771,179.541,6.177,149.250
C08750=1144.447,-13.804,-47.759,179.539,6.177,149.251
C08751=1144.452,-14.053,-47.746,179.536,6.176,149.251
C08752=1144.457,-14.302,-47.734,179.534,6.175,149.252
C08753=1144.463,-14.552,-47.721,179.532,6.175,149.252
C08754=1144.469,-14.802,-47.709,179.529,6.174,149.253
C08755=1144.473,-15.052,-47.696,179.527,6.174,149.254
C08756=1144.478,-15.301,-47.683,179.525,6.173,149.254
C08757=1144.483,-15.551,-47.671,179.522,6.172,149.255
C08758=1144.489,-15.801,-47.659,179.520,6.172,149.255
C08759=1144.494,-16.050,-47.646,179.518,6.171,149.256
C08760=1144.499,-16.299,-47.634,179.514,6.170,149.256
C08761=1144.504,-16.550,-47.621,179.512,6.169,149.257
C08762=1144.509,-16.799,-47.609,179.510,6.168,149.257
C08763=1144.514,-17.049,-47.596,179.507,6.168,149.258
C08764=1144.520,-17.298,-47.584,179.505,6.167,149.259
C08765=1144.525,-17.548,-47.572,179.502,6.166,149.259
C08766=1144.530,-17.797,-47.559,179.500,6.166,149.260
C08767=1144.535,-18.047,-47.547,179.498,6.165,149.260
C08768=1144.540,-18.296,-47.535,179.495,6.164,149.261
C08769=1144.545,-18.546,-47.522,179.493,6.164,149.261
C08770=1144.551,-18.797,-47.509,179.491,6.163,149.262
C08771=1144.556,-19.046,-47.496,179.488,6.162,149.262
C08772=1144.562,-19.296,-47.485,179.486,6.162,149.263
C08773=1144.567,-19.545,-47.472,179.484,6.161,149.264
C08774=1144.572,-19.795,-47.459,179.481,6.160,149.264
C08775=1144.577,-20.044,-47.448,179.478,6.159,149.265
C08776=1144.582,-20.293,-47.435,179.476,6.158,149.265
C08777=1144.587,-20.543,-47.424,179.473,6.158,149.266
C08778=1144.592,-20.793,-47.411,179.471,6.157,149.266
C08779=1144.598,-21.043,-47.399,179.469,6.156,149.267
C08780=1144.602,-21.293,-47.386,179.466,6.156,149.268
C08781=1144.608,-21.543,-47.374,179.464,6.155,149.268
C08782=1144.613,-21.792,-47.362,179.461,6.155,149.269
C08783=1144.618,-22.042,-47.350,179.459,6.154,149.269
C08784=1144.623,-22.291,-47.337,179.457,6.153,149.270
C08785=1144.629,-22.541,-47.325,179.454,6.153,149.270
C08786=1144.634,-22.790,-47.313,179.452,6.152,149.271
C08787=1144.639,-23.040,-47.301,179.450,6.151,149.272
C08788=1144.644,-23.290,-47.288,179.447,6.151,149.272
C08789=1144.650,-23.540,-47.276,179.445,6.150,149.273
C08790=1144.655,-23.789,-47.264,179.443,6.149,149.273
C08791=1144.660,-24.039,-47.252,179.440,6.149,149.274
C08792=1144.666,-24.309,-47.239,179.438,6.148,149.274
C08793=1144.671,-24.578,-47.226,179.434,6.147,149.275
C08794=1144.677,-24.849,-47.213,179.432,6.146,149.276
C08795=1144.682,-25.119,-47.200,179.430,6.146,149.276
C08796=1144.687,-25.369,-47.188,179.427,6.145,149.277
C08797=1144.692,-25.618,-47.175,179.425,6.145,149.277
C08798=1144.698,-25.868,-47.163,179.423,6.144,149.278
C08799=1144.703,-26.118,-47.151,179.420,6.143,149.278
C08800=1144.708,-26.367,-47.139,179.418,6.143,149.279
C08801=1144.713,-26.617,-47.127,179.416,6.142,149.280
C08802=1144.718,-26.866,-47.115,179.413,6.141,149.280
C08803=1144.724,-27.116,-47.103,179.411,6.141,149.281
C08804=1144.729,-27.366,-47.091,179.409,6.140,149.281
C08805=1144.734,-27.616,-47.078,179.406,6.139,149.282
C08806=1144.740,-27.864,-47.068,179.404,6.139,149.282
C08807=1144.745,-28.114,-47.056,179.401,6.138,149.283
C08808=1144.750,-28.364,-47.043,179.399,6.137,149.284
C08809=1144.756,-28.614,-47.031,179.397,6.137,149.284
C08810=1144.761,-28.864,-47.019,179.394,6.136,149.285
C08811=1144.766,-29.113,-47.008,179.392,6.135,149.285
C08812=1144.771,-29.363,-46.995,179.389,6.135,149.286
C08813=1144.776,-29.612,-46.984,179.387,6.134,149.286
C08814=1144.782,-29.862,-46.972,179.385,6.133,149.287
C08815=1144.786,-30.112,-46.960,179.382,6.133,149.288
C08816=1144.791,-30.361,-46.948,179.380,6.132,149.288
C08817=1144.797,-30.611,-46.936,179.377,6.132,149.289
C08818=1144.802,-30.861,-46.924,179.375,6.131,149.289
C08819=1144.807,-31.111,-46.913,179.373,6.130,149.290
C08820=1144.812,-31.361,-46.901,179.370,6.130,149.290
C08821=1144.818,-31.610,-46.888,179.368,6.129,149.291
C08822=1144.822,-31.860,-46.877,179.365,6.129,149.292
C08823=1144.828,-32.109,-46.865,179.363,6.128,149.292
C08824=1144.834,-32.359,-46.854,179.361,6.127,149.292
C08825=1144.839,-32.609,-46.842,179.358,6.127,149.293
C08826=1144.844,-32.858,-46.830,179.356,6.126,149.294
C08827=1144.849,-33.108,-46.818,179.353,6.125,149.294
C08828=1144.854,-33.358,-46.806,179.351,6.125,149.295
C08829=1144.859,-33.607,-46.795,179.349,6.124,149.295
C08830=1144.865,-33.857,-46.783,179.346,6.124,149.296
C08831=1144.870,-34.107,-46.771,179.344,6.123,149.296
C08832=1144.875,-34.356,-46.760,179.342,6.122,149.297
C08833=1144.881,-34.606,-46.748,179.339,6.122,149.298
C08834=1144.886,-34.855,-46.735,179.337,6.121,149.298
C08835=1144.890,-35.105,-46.724,179.335,6.120,149.299
C08836=1144.896,-35.355,-46.712,179.332,6.120,149.299
C08837=1144.901,-35.605,-46.701,179.330,6.119,149.300
C08838=1144.906,-35.855,-46.689,179.328,6.118,149.300
C08839=1144.912,-36.104,-46.678,179.325,6.118,149.301
C08840=1144.917,-36.353,-46.666,179.323,6.117,149.302
C08841=1144.922,-36.603,-46.654,179.321,6.116,149.302
C08842=1144.927,-36.853,-46.643,179.318,6.117,149.303
C08843=1144.932,-37.103,-46.631,179.316,6.116,149.303
C08844=1144.938,-37.353,-46.619,179.314,6.115,149.304
C08845=1144.943,-37.602,-46.608,179.311,6.115,149.304
C08846=1144.948,-37.852,-46.596,179.309,6.114,149.305
C08847=1144.953,-38.101,-46.585,179.307,6.113,149.305
C08848=1144.959,-38.351,-46.573,179.304,6.113,149.306
C08849=1144.964,-38.601,-46.561,179.302,6.112,149.307
C08850=1144.969,-38.850,-46.550,179.300,6.112,149.307
C08851=1144.975,-39.100,-46.539,179.297,6.111,149.308
C08852=1144.979,-39.350,-46.527,179.295,6.110,149.308
C08853=1144.985,-39.600,-46.515,179.292,6.110,149.309
C08854=1144.990,-39.849,-46.504,179.290,6.109,149.309
C08855=1144.996,-40.098,-46.493,179.288,6.108,149.310
C08856=1145.000,-40.348,-46.481,179.285,6.108,149.311
C08857=1145.006,-40.599,-46.470,179.283,6.107,149.311
C08858=1145.011,-40.848,-46.459,179.281,6.106,149.312
C08859=1145.017,-41.098,-46.447,179.278,6.106,149.312
C08860=1145.021,-41.347,-46.436,179.277,6.106,149.313
C08861=1145.027,-41.597,-46.424,179.274,6.105,149.313
C08862=1145.032,-41.847,-46.413,179.272,6.104,149.314
C08863=1145.038,-42.096,-46.401,179.269,6.104,149.315
C08864=1145.042,-42.346,-46.390,179.267,6.103,149.315
C08865=1145.048,-42.596,-46.378,179.265,6.103,149.316
C08866=1145.053,-42.846,-46.368,179.262,6.102,149.316
C08867=1145.059,-43.095,-46.356,179.260,6.101,149.317
C08868=1145.063,-43.345,-46.345,179.257,6.101,149.317
C08869=1145.069,-43.595,-46.333,179.255,6.100,149.318
C08870=1145.074,-43.844,-46.322,179.253,6.099,149.318
C08871=1145.080,-44.094,-46.311,179.250,6.099,149.319
C08872=1145.085,-44.344,-46.300,179.249,6.099,149.320
C08873=1145.089,-44.593,-46.288,179.247,6.098,149.320
C08874=1145.095,-44.843,-46.277,179.244,6.098,149.321
C08875=1145.100,-45.092,-46.265,179.242,6.097,149.321
C08876=1145.106,-45.343,-46.254,179.239,6.097,149.322
C08877=1145.110,-45.592,-46.243,179.237,6.096,149.322
C08878=1145.116,-45.841,-46.232,179.235,6.095,149.323
C08879=1145.121,-46.091,-46.220,179.232,6.095,149.324
C08880=1145.126,-46.341,-46.210,179.230,6.094,149.324
C08881=1145.132,-46.591,-46.198,179.228,6.093,149.325
C08882=1145.137,-46.840,-46.187,179.225,6.093,149.325
C08883=1145.142,-47.090,-46.175,179.223,6.093,149.326
C08884=1145.148,-47.340,-46.165,179.221,6.092,149.326
C08885=1145.153,-47.589,-46.153,179.219,6.092,149.327
C08886=1145.157,-47.839,-46.142,179.216,6.091,149.327
C08887=1145.164,-48.089,-46.131,179.214,6.090,149.328
C08888=1145.168,-48.338,-46.120,179.212,6.090,149.329
C08889=1145.173,-48.588,-46.109,179.209,6.089,149.329
C08890=1145.179,-48.838,-46.098,179.207,6.088,149.330
C08891=1145.184,-49.088,-46.087,179.204,6.088,149.330
C08892=1145.189,-49.337,-46.075,179.203,6.088,149.331
C08893=1145.195,-49.587,-46.065,179.200,6.087,149.331
C08894=1145.200,-49.837,-46.053,179.198,6.086,149.332
C08895=1145.204,-50.086,-46.042,179.195,6.086,149.333
C08896=1145.211,-50.357,-46.030,179.193,6.085,149.333
C08897=1145.217,-50.628,-46.019,179.190,6.085,149.334
C08898=1145.223,-50.898,-46.007,179.188,6.084,149.334
C08899=1145.228,-51.169,-45.994,179.186,6.084,149.335
C08900=1145.233,-51.419,-45.983,179.183,6.083,149.335
C08901=1145.238,-51.668,-45.972,179.181,6.083,149.336
C08902=1145.243,-51.918,-45.962,179.179,6.082,149.337
C08903=1145.249,-52.168,-45.950,179.176,6.081,149.337
C08904=1145.254,-52.418,-45.940,179.174,6.081,149.338
C08905=1145.259,-52.667,-45.928,179.172,6.081,149.338
C08906=1145.265,-52.917,-45.918,179.170,6.080,149.339
C08907=1145.270,-53.167,-45.906,179.167,6.079,149.339
C08908=1145.275,-53.417,-45.896,179.165,6.079,149.340
C08909=1145.280,-53.666,-45.885,179.163,6.078,149.340
C08910=1145.285,-53.916,-45.874,179.160,6.077,149.341
C08911=1145.291,-54.165,-45.863,179.158,6.077,149.342
C08912=1145.296,-54.416,-45.852,179.156,6.077,149.342
C08913=1145.302,-54.665,-45.841,179.154,6.076,149.343
C08914=1145.307,-54.915,-45.830,179.152,6.076,149.343
C08915=1145.311,-55.165,-45.819,179.149,6.075,149.344
C08916=1145.318,-55.414,-45.808,179.147,6.074,149.344
C08917=1145.322,-55.664,-45.797,179.145,6.074,149.345
C08918=1145.328,-55.914,-45.787,179.142,6.073,149.346
C08919=1145.333,-56.163,-45.776,179.140,6.073,149.346
C08920=1145.338,-56.413,-45.765,179.138,6.072,149.347
C08921=1145.343,-56.662,-45.754,179.135,6.072,149.347
C08922=1145.349,-56.912,-45.743,179.133,6.071,149.348
C08923=1145.354,-57.162,-45.733,179.131,6.070,149.348
C08924=1145.359,-57.412,-45.721,179.128,6.070,149.349
C08925=1145.365,-57.662,-45.711,179.127,6.070,149.349
C08926=1145.369,-57.911,-45.700,179.125,6.069,149.350
C08927=1145.375,-58.161,-45.690,179.122,6.069,149.351
C08928=1145.380,-58.411,-45.679,179.120,6.068,149.351
C08929=1145.385,-58.660,-45.668,179.118,6.067,149.352
C08930=1145.391,-58.911,-45.657,179.115,6.067,149.352
C08931=1145.397,-59.160,-45.647,179.113,6.067,149.353
C08932=1145.401,-59.410,-45.636,179.111,6.066,149.353
C08933=1145.407,-59.659,-45.625,179.108,6.066,149.354
C08934=1145.412,-59.909,-45.615,179.106,6.065,149.354
C08935=1145.417,-60.158,-45.604,179.104,6.064,149.355
C08936=1145.422,-60.409,-45.593,179.101,6.064,149.356
C08937=1145.428,-60.658,-45.583,179.100,6.064,149.356
C08938=1145.432,-60.908,-45.572,179.098,6.063,149.357
C08939=1145.438,-61.157,-45.562,179.095,6.063,149.357
C08940=1145.443,-61.408,-45.551,179.093,6.062,149.358
C08941=1145.448,-61.657,-45.540,179.091,6.061,149.358
C08942=1145.453,-61.907,-45.529,179.088,6.061,149.359
C08943=1145.459,-62.156,-45.519,179.086,6.061,149.359
C08944=1145.465,-62.407,-45.508,179.084,6.060,149.360
C08945=1145.470,-62.656,-45.497,179.081,6.060,149.361
C08946=1145.476,-62.905,-45.487,179.079,6.059,149.361
C08947=1145.481,-63.156,-45.476,179.077,6.058,149.362
C08948=1145.486,-63.405,-45.466,179.075,6.059,149.362
C08949=1145.491,-63.655,-45.455,179.073,6.058,149.363
C08950=1145.496,-63.904,-45.445,179.071,6.057,149.363
C08951=1145.501,-64.155,-45.434,179.068,6.057,149.364
C08952=1145.507,-64.404,-45.424,179.066,6.056,149.364
C08953=1145.512,-64.654,-45.413,179.064,6.056,149.365
C08954=1145.517,-64.903,-45.402,179.061,6.055,149.366
C08955=1145.523,-65.153,-45.392,179.059,6.055,149.366
C08956=1145.528,-65.403,-45.382,179.057,6.054,149.367
C08957=1145.533,-65.653,-45.371,179.054,6.054,149.367
C08958=1145.538,-65.903,-45.361,179.053,6.054,149.368
C08959=1145.544,-66.152,-45.351,179.051,6.053,149.368
C08960=1145.549,-66.402,-45.341,179.048,6.052,149.369
C08961=1145.554,-66.651,-45.330,179.046,6.052,149.369
C08962=1145.559,-66.901,-45.320,179.044,6.051,149.370
C08963=1145.564,-67.151,-45.309,179.042,6.051,149.371
C08964=1145.570,-67.401,-45.299,179.039,6.051,149.371
C08965=1145.575,-67.650,-45.289,179.037,6.050,149.372
C08966=1145.580,-67.900,-45.278,179.034,6.049,149.372
C08967=1145.586,-68.150,-45.268,179.033,6.049,149.373
C08968=1145.591,-68.400,-45.257,179.031,6.049,149.373
C08969=1145.597,-68.650,-45.247,179.028,6.048,149.374
C08970=1145.602,-68.899,-45.236,179.026,6.047,149.374
C08971=1145.607,-69.149,-45.225,179.024,6.047,149.375
C08972=1145.613,-69.398,-45.215,179.022,6.047,149.376
C08973=1145.618,-69.648,-45.205,179.019,6.046,149.376
C08974=1145.622,-69.898,-45.195,179.017,6.046,149.377
C08975=1145.628,-70.147,-45.185,179.015,6.045,149.377
C08976=1145.634,-70.397,-45.175,179.013,6.045,149.378
C08977=1145.639,-70.647,-45.164,179.011,6.044,149.378
C08978=1145.644,-70.897,-45.154,179.009,6.044,149.379
C08979=1145.650,-71.146,-45.144,179.006,6.043,149.379
C08980=1145.655,-71.397,-45.133,179.004,6.043,149.380
C08981=1145.660,-71.646,-45.123,179.002,6.043,149.380
C08982=1145.665,-71.895,-45.113,178.999,6.042,149.381
C08983=1145.670,-72.146,-45.103,178.997,6.041,149.382
C08984=1145.676,-72.395,-45.092,178.995,6.041,149.382
C08985=1145.681,-72.645,-45.082,178.993,6.041,149.383
C08986=1145.686,-72.895,-45.072,178.991,6.040,149.383
C08987=1145.692,-73.144,-45.061,178.989,6.039,149.384
C08988=1145.697,-73.394,-45.053,178.986,6.039,149.384
C08989=1145.703,-73.644,-45.042,178.984,6.039,149.385
C08990=1145.708,-73.894,-45.032,178.982,6.038,149.385
C08991=1145.713,-74.144,-45.022,178.980,6.038,149.386
C08992=1145.719,-74.393,-45.011,178.977,6.037,149.387
C08993=1145.723,-74.643,-45.001,178.976,6.037,149.387
C08994=1145.729,-74.893,-44.991,178.973,6.036,149.388
C08995=1145.734,-75.142,-44.981,178.971,6.036,149.388
C08996=1145.740,-75.392,-44.971,178.969,6.035,149.389
C08997=1145.745,-75.642,-44.960,178.967,6.035,149.389
C08998=1145.750,-75.892,-44.951,178.965,6.035,149.390
C08999=1145.756,-76.141,-44.941,178.962,6.034,149.390
C09000=1145.762,-76.413,-44.930,178.960,6.033,149.391
C09001=1145.767,-76.684,-44.919,178.957,6.033,149.392
C09002=1145.773,-76.955,-44.907,178.956,6.033,149.392
C09003=1145.779,-77.227,-44.897,178.953,6.033,149.393
C09004=1145.785,-77.477,-44.887,178.951,6.032,149.393
C09005=1145.789,-77.726,-44.877,178.949,6.031,149.394
C09006=1145.794,-77.976,-44.867,178.946,6.030,149.394
C09007=1145.800,-78.226,-44.857,178.944,6.031,149.395
C09008=1145.806,-78.476,-44.847,178.942,6.030,149.395
C09009=1145.811,-78.725,-44.838,178.940,6.029,149.396
C09010=1145.816,-78.975,-44.827,178.938,6.030,149.397
C09011=1145.821,-79.225,-44.817,178.936,6.029,149.397
C09012=1145.826,-79.475,-44.808,178.934,6.028,149.398
C09013=1145.832,-79.724,-44.798,178.931,6.027,149.398
C09014=1145.838,-79.974,-44.787,178.929,6.028,149.399
C09015=1145.843,-80.224,-44.777,178.927,6.027,149.399
C09016=1145.848,-80.474,-44.768,178.925,6.026,149.400
C09017=1145.853,-80.723,-44.758,178.923,6.026,149.400
C09018=1145.859,-80.973,-44.748,178.921,6.026,149.401
C09019=1145.864,-81.222,-44.738,178.918,6.025,149.401
C09020=1145.869,-81.473,-44.728,178.916,6.024,149.402
C09021=1145.874,-81.722,-44.718,178.914,6.025,149.403
C09022=1145.880,-81.972,-44.708,178.912,6.024,149.403
C09023=1145.886,-82.222,-44.699,178.910,6.023,149.404
C09024=1145.890,-82.471,-44.689,178.908,6.023,149.404
C09025=1145.895,-82.721,-44.679,178.905,6.023,149.405
C09026=1145.901,-82.972,-44.669,178.903,6.022,149.405
C09027=1145.906,-83.221,-44.659,178.901,6.021,149.406
C09028=1145.912,-83.470,-44.649,178.900,6.021,149.406
C09029=1145.917,-83.720,-44.640,178.897,6.021,149.407
C09030=1145.923,-83.970,-44.630,178.895,6.020,149.407
C09031=1145.928,-84.220,-44.620,178.893,6.020,149.408
C09032=1145.933,-84.470,-44.611,178.891,6.020,149.408
C09033=1145.938,-84.719,-44.600,178.888,6.019,149.409
C09034=1145.943,-84.969,-44.591,178.886,6.018,149.410
C09035=1145.949,-85.219,-44.581,178.884,6.018,149.410
C09036=1145.955,-85.468,-44.571,178.882,6.018,149.411
C09037=1145.960,-85.718,-44.562,178.880,6.017,149.411
C09038=1145.965,-85.968,-44.552,178.878,6.017,149.412
C09039=1145.970,-86.218,-44.542,178.876,6.017,149.412
C09040=1145.976,-86.468,-44.533,178.873,6.016,149.413
C09041=1145.980,-86.717,-44.523,178.871,6.016,149.413
C09042=1145.986,-86.967,-44.513,178.869,6.015,149.414
C09043=1145.991,-87.216,-44.504,178.867,6.015,149.414
C09044=1145.997,-87.467,-44.494,178.865,6.015,149.415
C09045=1146.002,-87.716,-44.485,178.863,6.014,149.416
C09046=1146.007,-87.967,-44.475,178.861,6.014,149.416
C09047=1146.012,-88.216,-44.465,178.859,6.014,149.417
C09048=1146.018,-88.466,-44.456,178.857,6.013,149.417
C09049=1146.023,-88.715,-44.446,178.854,6.013,149.418
C09050=1146.029,-88.965,-44.436,178.853,6.013,149.418
C09051=1146.034,-89.215,-44.427,178.850,6.012,149.419
C09052=1146.039,-89.464,-44.417,178.848,6.011,149.419
C09053=1146.044,-89.714,-44.408,178.845,6.011,149.420
C09054=1146.050,-89.964,-44.398,178.844,6.011,149.420
C09055=1146.055,-90.214,-44.389,178.842,6.010,149.421
C09056=1146.061,-90.464,-44.379,178.840,6.009,149.421
C09057=1146.065,-90.714,-44.369,178.837,6.010,149.422
C09058=1146.071,-90.964,-44.360,178.835,6.009,149.423
C09059=1146.076,-91.213,-44.350,178.833,6.008,149.423
C09060=1146.082,-91.463,-44.341,178.831,6.008,149.424
C09061=1146.087,-91.712,-44.331,178.829,6.008,149.424
C09062=1146.093,-91.963,-44.322,178.827,6.008,149.425
C09063=1146.098,-92.212,-44.313,178.825,6.007,149.425
C09064=1146.103,-92.462,-44.303,178.823,6.006,149.426
C09065=1146.109,-92.712,-44.294,178.821,6.006,149.426
C09066=1146.114,-92.961,-44.284,178.819,6.006,149.427
C09067=1146.120,-93.211,-44.275,178.816,6.005,149.427
C09068=1146.125,-93.461,-44.266,178.815,6.005,149.428
C09069=1146.130,-93.711,-44.255,178.813,6.004,149.428
C09070=1146.135,-93.960,-44.247,178.810,6.004,149.429
C09071=1146.140,-94.210,-44.237,178.808,6.004,149.430
C09072=1146.146,-94.460,-44.227,178.806,6.003,149.430
C09073=1146.151,-94.710,-44.219,178.804,6.003,149.431
C09074=1146.157,-94.959,-44.208,178.802,6.003,149.431
C09075=1146.162,-95.209,-44.199,178.800,6.002,149.432
C09076=1146.167,-95.459,-44.191,178.797,6.001,149.432
C09077=1146.173,-95.709,-44.180,178.796,6.001,149.433
C09078=1146.178,-95.958,-44.171,178.794,6.001,149.433
C09079=1146.183,-96.208,-44.163,178.791,6.000,149.434
C09080=1146.189,-96.458,-44.152,178.789,6.000,149.434
C09081=1146.194,-96.708,-44.143,178.787,6.000,149.435
C09082=1146.199,-96.957,-44.135,178.786,6.000,149.435
C09083=1146.205,-97.208,-44.125,178.783,5.999,149.436
C09084=1146.210,-97.457,-44.115,178.781,5.999,149.437
C09085=1146.216,-97.707,-44.106,178.779,5.999,149.437
C09086=1146.221,-97.957,-44.097,178.777,5.998,149.437
C09087=1146.226,-98.206,-44.087,178.775,5.997,149.438
C09088=1146.231,-98.456,-44.079,178.773,5.997,149.438
C09089=1146.237,-98.706,-44.069,178.770,5.997,149.439
C09090=1146.242,-98.956,-44.060,178.768,5.996,149.440
C09091=1146.247,-99.206,-44.051,178.767,5.996,149.440
C09092=1146.253,-99.455,-44.041,178.764,5.995,149.441
C09093=1146.258,-99.705,-44.032,178.763,5.995,149.441
C09094=1146.263,-99.955,-44.023,178.760,5.995,149.442
C09095=1146.269,-100.205,-44.014,178.758,5.994,149.442
C09096=1146.274,-100.454,-44.004,178.756,5.994,149.443
C09097=1146.280,-100.704,-43.996,178.754,5.993,149.443
C09098=1146.285,-100.953,-43.987,178.752,5.993,149.444
C09099=1146.291,-101.204,-43.977,178.750,5.993,149.444
C09100=1146.296,-101.453,-43.968,178.748,5.992,149.445
C09101=1146.301,-101.703,-43.959,178.746,5.992,149.445
C09102=1146.306,-101.953,-43.950,178.744,5.992,149.446
C09103=1146.312,-102.203,-43.940,178.742,5.991,149.446
C09104=1146.318,-102.475,-43.931,178.740,5.991,149.447
C09105=1146.323,-102.747,-43.921,178.737,5.991,149.448
C09106=1146.329,-103.020,-43.911,178.735,5.990,149.448
C09107=1146.335,-103.291,-43.901,178.733,5.989,149.449
C09108=1146.340,-103.541,-43.892,178.731,5.989,149.449
C09109=1146.346,-103.791,-43.883,178.729,5.989,149.450
C09110=1146.351,-104.041,-43.874,178.727,5.989,149.450
C09111=1146.357,-104.291,-43.865,178.725,5.988,149.451
C09112=1146.362,-104.541,-43.856,178.722,5.988,149.451
C09113=1146.367,-104.790,-43.846,178.721,5.988,149.452
C09114=1146.372,-105.040,-43.837,178.719,5.987,149.452
C09115=1146.378,-105.290,-43.828,178.717,5.987,149.453
C09116=1146.383,-105.539,-43.820,178.715,5.986,149.453
C09117=1146.389,-105.789,-43.811,178.713,5.985,149.454
C09118=1146.394,-106.039,-43.802,178.710,5.986,149.455
C09119=1146.399,-106.288,-43.793,178.708,5.985,149.455
C09120=1146.405,-106.539,-43.783,178.707,5.985,149.456
C09121=1146.410,-106.788,-43.774,178.705,5.984,149.456
C09122=1146.415,-107.038,-43.766,178.702,5.984,149.457
C09123=1146.421,-107.287,-43.757,178.701,5.984,149.457
C09124=1146.426,-107.537,-43.748,178.698,5.983,149.458
C09125=1146.431,-107.787,-43.739,178.696,5.983,149.458
C09126=1146.436,-108.037,-43.730,178.694,5.983,149.459
C09127=1146.442,-108.287,-43.721,178.692,5.982,149.459
C09128=1146.447,-108.537,-43.712,178.690,5.982,149.460
C09129=1146.453,-108.787,-43.703,178.688,5.981,149.460
C09130=1146.458,-109.036,-43.695,178.687,5.981,149.461
C09131=1146.464,-109.286,-43.686,178.684,5.981,149.461
C09132=1146.469,-109.536,-43.677,178.682,5.981,149.462
C09133=1146.474,-109.786,-43.668,178.680,5.980,149.462
C09134=1146.479,-110.035,-43.659,178.678,5.979,149.463
C09135=1146.486,-110.285,-43.650,178.676,5.979,149.463
C09136=1146.491,-110.535,-43.641,178.674,5.979,149.464
C09137=1146.496,-110.785,-43.632,178.673,5.979,149.464
C09138=1146.501,-111.034,-43.623,178.670,5.978,149.465
C09139=1146.506,-111.284,-43.614,178.668,5.978,149.466
C09140=1146.512,-111.534,-43.606,178.666,5.978,149.466
C09141=1146.517,-111.784,-43.598,178.664,5.977,149.466
C09142=1146.523,-112.034,-43.589,178.662,5.977,149.467
C09143=1146.528,-112.284,-43.580,178.660,5.976,149.467
C09144=1146.533,-112.534,-43.571,178.659,5.976,149.468
C09145=1146.539,-112.783,-43.562,178.656,5.976,149.469
C09146=1146.544,-113.032,-43.553,178.654,5.976,149.469
C09147=1146.549,-113.282,-43.544,178.652,5.975,149.470
C09148=1146.555,-113.533,-43.536,178.650,5.974,149.470
